Fanuc TP program (LS listing): FM112728.ls

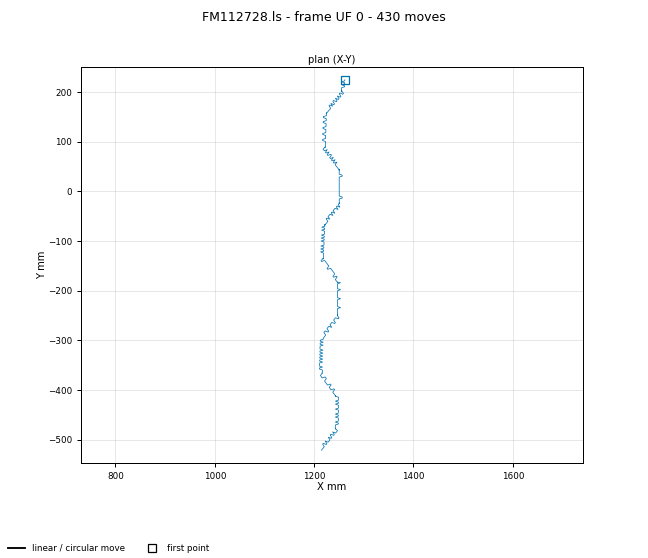
[picture p0: tool path of FM112728.ls in frame UF 0, 430 of 430 moves have a stored position in this frame; points joined in program order, loops and branches not executed]
/PROG  FM112728
/ATTR
OWNER		= MNEDITOR;
COMMENT		= "Auto FANUC move";
PROG_SIZE	= 0;
CREATE		= DATE 26-05-06  TIME 11:27:28;
MODIFIED	= DATE 26-05-06  TIME 11:27:28;
FILE_NAME	= ;
VERSION		= 0;
LINE_COUNT	= 435;
MEMORY_SIZE	= 0;
PROTECT		= READ_WRITE;
TCD:  STACK_SIZE	= 0,
      TASK_PRIORITY	= 50,
      TIME_SLICE	= 0,
      BUSY_LAMP_OFF	= 0,
      ABORT_REQUEST	= 0,
      PAUSE_REQUEST	= 0;
DEFAULT_GROUP	= 1,*,*,*,*;
CONTROL_CODE	= 00000000 00000000;
/MN
   1:  UFRAME_NUM=0 ;
   2:  UTOOL_NUM=1 ;
   3:  R[93]=10 ;
   4:  L P[1] 7mm/sec FINE ;
   5:  L P[2] 7mm/sec CNT50 ;
   6:  L P[3] 7mm/sec CNT50 ;
   7:  L P[4] 7mm/sec CNT50 ;
   8:  L P[5] 7mm/sec CNT50 ;
   9:  L P[6] 7mm/sec CNT50 ;
  10:  L P[7] 7mm/sec CNT50 ;
  11:  L P[8] 7mm/sec CNT50 ;
  12:  L P[9] 7mm/sec CNT50 ;
  13:  L P[10] 7mm/sec CNT50 ;
  14:  L P[11] 7mm/sec CNT50 ;
  15:  L P[12] 7mm/sec CNT50 ;
  16:  L P[13] 7mm/sec CNT50 ;
  17:  L P[14] 7mm/sec CNT50 ;
  18:  L P[15] 7mm/sec CNT50 ;
  19:  L P[16] 7mm/sec CNT50 ;
  20:  L P[17] 7mm/sec CNT50 ;
  21:  L P[18] 7mm/sec CNT50 ;
  22:  L P[19] 7mm/sec CNT50 ;
  23:  L P[20] 7mm/sec CNT50 ;
  24:  L P[21] 7mm/sec CNT50 ;
  25:  L P[22] 7mm/sec CNT50 ;
  26:  L P[23] 7mm/sec CNT50 ;
  27:  L P[24] 7mm/sec CNT50 ;
  28:  L P[25] 7mm/sec CNT50 ;
  29:  L P[26] 7mm/sec CNT50 ;
  30:  L P[27] 7mm/sec CNT50 ;
  31:  L P[28] 7mm/sec CNT50 ;
  32:  L P[29] 7mm/sec CNT50 ;
  33:  L P[30] 7mm/sec CNT50 ;
  34:  L P[31] 7mm/sec CNT50 ;
  35:  L P[32] 7mm/sec CNT50 ;
  36:  L P[33] 7mm/sec CNT50 ;
  37:  L P[34] 7mm/sec CNT50 ;
  38:  L P[35] 7mm/sec CNT50 ;
  39:  L P[36] 7mm/sec CNT50 ;
  40:  L P[37] 7mm/sec CNT50 ;
  41:  L P[38] 7mm/sec CNT50 ;
  42:  L P[39] 7mm/sec CNT50 ;
  43:  L P[40] 7mm/sec CNT50 ;
  44:  L P[41] 7mm/sec CNT50 ;
  45:  L P[42] 7mm/sec CNT50 ;
  46:  L P[43] 7mm/sec CNT50 ;
  47:  L P[44] 7mm/sec CNT50 ;
  48:  L P[45] 7mm/sec CNT50 ;
  49:  L P[46] 7mm/sec CNT50 ;
  50:  L P[47] 7mm/sec CNT50 ;
  51:  L P[48] 7mm/sec CNT50 ;
  52:  L P[49] 7mm/sec CNT50 ;
  53:  L P[50] 7mm/sec CNT50 ;
  54:  L P[51] 7mm/sec CNT50 ;
  55:  L P[52] 7mm/sec CNT50 ;
  56:  L P[53] 7mm/sec CNT50 ;
  57:  L P[54] 7mm/sec CNT50 ;
  58:  L P[55] 7mm/sec CNT50 ;
  59:  L P[56] 7mm/sec CNT50 ;
  60:  L P[57] 7mm/sec CNT50 ;
  61:  L P[58] 7mm/sec CNT50 ;
  62:  L P[59] 7mm/sec CNT50 ;
  63:  L P[60] 7mm/sec CNT50 ;
  64:  L P[61] 7mm/sec CNT50 ;
  65:  L P[62] 7mm/sec CNT50 ;
  66:  L P[63] 7mm/sec CNT50 ;
  67:  L P[64] 7mm/sec CNT50 ;
  68:  L P[65] 7mm/sec CNT50 ;
  69:  L P[66] 7mm/sec CNT50 ;
  70:  L P[67] 7mm/sec CNT50 ;
  71:  L P[68] 7mm/sec CNT50 ;
  72:  L P[69] 7mm/sec CNT50 ;
  73:  L P[70] 7mm/sec CNT50 ;
  74:  L P[71] 7mm/sec CNT50 ;
  75:  L P[72] 7mm/sec CNT50 ;
  76:  L P[73] 7mm/sec CNT50 ;
  77:  L P[74] 7mm/sec CNT50 ;
  78:  L P[75] 7mm/sec CNT50 ;
  79:  L P[76] 7mm/sec CNT50 ;
  80:  L P[77] 7mm/sec CNT50 ;
  81:  L P[78] 7mm/sec CNT50 ;
  82:  L P[79] 7mm/sec CNT50 ;
  83:  L P[80] 7mm/sec CNT50 ;
  84:  L P[81] 7mm/sec CNT50 ;
  85:  L P[82] 7mm/sec CNT50 ;
  86:  L P[83] 7mm/sec CNT50 ;
  87:  L P[84] 7mm/sec CNT50 ;
  88:  L P[85] 7mm/sec CNT50 ;
  89:  L P[86] 7mm/sec CNT50 ;
  90:  L P[87] 7mm/sec CNT50 ;
  91:  L P[88] 7mm/sec CNT50 ;
  92:  L P[89] 7mm/sec CNT50 ;
  93:  L P[90] 7mm/sec CNT50 ;
  94:  L P[91] 7mm/sec CNT50 ;
  95:  L P[92] 7mm/sec CNT50 ;
  96:  L P[93] 7mm/sec CNT50 ;
  97:  L P[94] 7mm/sec CNT50 ;
  98:  L P[95] 7mm/sec CNT50 ;
  99:  L P[96] 7mm/sec CNT50 ;
 100:  L P[97] 7mm/sec CNT50 ;
 101:  L P[98] 7mm/sec CNT50 ;
 102:  L P[99] 7mm/sec CNT50 ;
 103:  L P[100] 7mm/sec CNT50 ;
 104:  L P[101] 7mm/sec CNT50 ;
 105:  L P[102] 7mm/sec CNT50 ;
 106:  L P[103] 7mm/sec CNT50 ;
 107:  L P[104] 7mm/sec CNT50 ;
 108:  L P[105] 7mm/sec CNT50 ;
 109:  L P[106] 7mm/sec CNT50 ;
 110:  L P[107] 7mm/sec CNT50 ;
 111:  L P[108] 7mm/sec CNT50 ;
 112:  L P[109] 7mm/sec CNT50 ;
 113:  L P[110] 7mm/sec CNT50 ;
 114:  L P[111] 7mm/sec CNT50 ;
 115:  L P[112] 7mm/sec CNT50 ;
 116:  L P[113] 7mm/sec CNT50 ;
 117:  L P[114] 7mm/sec CNT50 ;
 118:  L P[115] 7mm/sec CNT50 ;
 119:  L P[116] 7mm/sec CNT50 ;
 120:  L P[117] 7mm/sec CNT50 ;
 121:  L P[118] 7mm/sec CNT50 ;
 122:  L P[119] 7mm/sec CNT50 ;
 123:  L P[120] 7mm/sec CNT50 ;
 124:  L P[121] 7mm/sec CNT50 ;
 125:  L P[122] 7mm/sec CNT50 ;
 126:  L P[123] 7mm/sec CNT50 ;
 127:  L P[124] 7mm/sec CNT50 ;
 128:  L P[125] 7mm/sec CNT50 ;
 129:  L P[126] 7mm/sec CNT50 ;
 130:  L P[127] 7mm/sec CNT50 ;
 131:  L P[128] 7mm/sec CNT50 ;
 132:  L P[129] 7mm/sec CNT50 ;
 133:  L P[130] 7mm/sec CNT50 ;
 134:  L P[131] 7mm/sec CNT50 ;
 135:  L P[132] 7mm/sec CNT50 ;
 136:  L P[133] 7mm/sec CNT50 ;
 137:  L P[134] 7mm/sec CNT50 ;
 138:  L P[135] 7mm/sec CNT50 ;
 139:  L P[136] 7mm/sec CNT50 ;
 140:  L P[137] 7mm/sec CNT50 ;
 141:  L P[138] 7mm/sec CNT50 ;
 142:  L P[139] 7mm/sec CNT50 ;
 143:  L P[140] 7mm/sec CNT50 ;
 144:  L P[141] 7mm/sec CNT50 ;
 145:  L P[142] 7mm/sec CNT50 ;
 146:  L P[143] 7mm/sec CNT50 ;
 147:  L P[144] 7mm/sec CNT50 ;
 148:  L P[145] 7mm/sec CNT50 ;
 149:  L P[146] 7mm/sec CNT50 ;
 150:  L P[147] 7mm/sec CNT50 ;
 151:  L P[148] 7mm/sec CNT50 ;
 152:  L P[149] 7mm/sec CNT50 ;
 153:  L P[150] 7mm/sec CNT50 ;
 154:  L P[151] 7mm/sec CNT50 ;
 155:  L P[152] 7mm/sec CNT50 ;
 156:  L P[153] 7mm/sec CNT50 ;
 157:  L P[154] 7mm/sec CNT50 ;
 158:  L P[155] 7mm/sec CNT50 ;
 159:  L P[156] 7mm/sec CNT50 ;
 160:  L P[157] 7mm/sec CNT50 ;
 161:  L P[158] 7mm/sec CNT50 ;
 162:  L P[159] 7mm/sec CNT50 ;
 163:  L P[160] 7mm/sec CNT50 ;
 164:  L P[161] 7mm/sec CNT50 ;
 165:  L P[162] 7mm/sec CNT50 ;
 166:  L P[163] 7mm/sec CNT50 ;
 167:  L P[164] 7mm/sec CNT50 ;
 168:  L P[165] 7mm/sec CNT50 ;
 169:  L P[166] 7mm/sec CNT50 ;
 170:  L P[167] 7mm/sec CNT50 ;
 171:  L P[168] 7mm/sec CNT50 ;
 172:  L P[169] 7mm/sec CNT50 ;
 173:  L P[170] 7mm/sec CNT50 ;
 174:  L P[171] 7mm/sec CNT50 ;
 175:  L P[172] 7mm/sec CNT50 ;
 176:  L P[173] 7mm/sec CNT50 ;
 177:  L P[174] 7mm/sec CNT50 ;
 178:  L P[175] 7mm/sec CNT50 ;
 179:  L P[176] 7mm/sec CNT50 ;
 180:  L P[177] 7mm/sec CNT50 ;
 181:  L P[178] 7mm/sec CNT50 ;
 182:  L P[179] 7mm/sec CNT50 ;
 183:  L P[180] 7mm/sec CNT50 ;
 184:  L P[181] 7mm/sec CNT50 ;
 185:  L P[182] 7mm/sec CNT50 ;
 186:  L P[183] 7mm/sec CNT50 ;
 187:  L P[184] 7mm/sec CNT50 ;
 188:  L P[185] 7mm/sec CNT50 ;
 189:  L P[186] 7mm/sec CNT50 ;
 190:  L P[187] 7mm/sec CNT50 ;
 191:  L P[188] 7mm/sec CNT50 ;
 192:  L P[189] 7mm/sec CNT50 ;
 193:  L P[190] 7mm/sec CNT50 ;
 194:  L P[191] 7mm/sec CNT50 ;
 195:  L P[192] 7mm/sec CNT50 ;
 196:  L P[193] 7mm/sec CNT50 ;
 197:  L P[194] 7mm/sec CNT50 ;
 198:  L P[195] 7mm/sec CNT50 ;
 199:  L P[196] 7mm/sec CNT50 ;
 200:  L P[197] 7mm/sec CNT50 ;
 201:  L P[198] 7mm/sec CNT50 ;
 202:  L P[199] 7mm/sec CNT50 ;
 203:  L P[200] 7mm/sec CNT50 ;
 204:  L P[201] 7mm/sec CNT50 ;
 205:  L P[202] 7mm/sec CNT50 ;
 206:  L P[203] 7mm/sec CNT50 ;
 207:  L P[204] 7mm/sec CNT50 ;
 208:  L P[205] 7mm/sec CNT50 ;
 209:  L P[206] 7mm/sec CNT50 ;
 210:  L P[207] 7mm/sec CNT50 ;
 211:  L P[208] 7mm/sec CNT50 ;
 212:  L P[209] 7mm/sec CNT50 ;
 213:  L P[210] 7mm/sec CNT50 ;
 214:  L P[211] 7mm/sec CNT50 ;
 215:  L P[212] 7mm/sec CNT50 ;
 216:  L P[213] 7mm/sec CNT50 ;
 217:  L P[214] 7mm/sec CNT50 ;
 218:  L P[215] 7mm/sec CNT50 ;
 219:  L P[216] 7mm/sec CNT50 ;
 220:  L P[217] 7mm/sec CNT50 ;
 221:  L P[218] 7mm/sec CNT50 ;
 222:  L P[219] 7mm/sec CNT50 ;
 223:  L P[220] 7mm/sec CNT50 ;
 224:  L P[221] 7mm/sec CNT50 ;
 225:  L P[222] 7mm/sec CNT50 ;
 226:  L P[223] 7mm/sec CNT50 ;
 227:  L P[224] 7mm/sec CNT50 ;
 228:  L P[225] 7mm/sec CNT50 ;
 229:  L P[226] 7mm/sec CNT50 ;
 230:  L P[227] 7mm/sec CNT50 ;
 231:  L P[228] 7mm/sec CNT50 ;
 232:  L P[229] 7mm/sec CNT50 ;
 233:  L P[230] 7mm/sec CNT50 ;
 234:  L P[231] 7mm/sec CNT50 ;
 235:  L P[232] 7mm/sec CNT50 ;
 236:  L P[233] 7mm/sec CNT50 ;
 237:  L P[234] 7mm/sec CNT50 ;
 238:  L P[235] 7mm/sec CNT50 ;
 239:  L P[236] 7mm/sec CNT50 ;
 240:  L P[237] 7mm/sec CNT50 ;
 241:  L P[238] 7mm/sec CNT50 ;
 242:  L P[239] 7mm/sec CNT50 ;
 243:  L P[240] 7mm/sec CNT50 ;
 244:  L P[241] 7mm/sec CNT50 ;
 245:  L P[242] 7mm/sec CNT50 ;
 246:  L P[243] 7mm/sec CNT50 ;
 247:  L P[244] 7mm/sec CNT50 ;
 248:  L P[245] 7mm/sec CNT50 ;
 249:  L P[246] 7mm/sec CNT50 ;
 250:  L P[247] 7mm/sec CNT50 ;
 251:  L P[248] 7mm/sec CNT50 ;
 252:  L P[249] 7mm/sec CNT50 ;
 253:  L P[250] 7mm/sec CNT50 ;
 254:  L P[251] 7mm/sec CNT50 ;
 255:  L P[252] 7mm/sec CNT50 ;
 256:  L P[253] 7mm/sec CNT50 ;
 257:  L P[254] 7mm/sec CNT50 ;
 258:  L P[255] 7mm/sec CNT50 ;
 259:  L P[256] 7mm/sec CNT50 ;
 260:  L P[257] 7mm/sec CNT50 ;
 261:  L P[258] 7mm/sec CNT50 ;
 262:  L P[259] 7mm/sec CNT50 ;
 263:  L P[260] 7mm/sec CNT50 ;
 264:  L P[261] 7mm/sec CNT50 ;
 265:  L P[262] 7mm/sec CNT50 ;
 266:  L P[263] 7mm/sec CNT50 ;
 267:  L P[264] 7mm/sec CNT50 ;
 268:  L P[265] 7mm/sec CNT50 ;
 269:  L P[266] 7mm/sec CNT50 ;
 270:  L P[267] 7mm/sec CNT50 ;
 271:  L P[268] 7mm/sec CNT50 ;
 272:  L P[269] 7mm/sec CNT50 ;
 273:  L P[270] 7mm/sec CNT50 ;
 274:  L P[271] 7mm/sec CNT50 ;
 275:  L P[272] 7mm/sec CNT50 ;
 276:  L P[273] 7mm/sec CNT50 ;
 277:  L P[274] 7mm/sec CNT50 ;
 278:  L P[275] 7mm/sec CNT50 ;
 279:  L P[276] 7mm/sec CNT50 ;
 280:  L P[277] 7mm/sec CNT50 ;
 281:  L P[278] 7mm/sec CNT50 ;
 282:  L P[279] 7mm/sec CNT50 ;
 283:  L P[280] 7mm/sec CNT50 ;
 284:  L P[281] 7mm/sec CNT50 ;
 285:  L P[282] 7mm/sec CNT50 ;
 286:  L P[283] 7mm/sec CNT50 ;
 287:  L P[284] 7mm/sec CNT50 ;
 288:  L P[285] 7mm/sec CNT50 ;
 289:  L P[286] 7mm/sec CNT50 ;
 290:  L P[287] 7mm/sec CNT50 ;
 291:  L P[288] 7mm/sec CNT50 ;
 292:  L P[289] 7mm/sec CNT50 ;
 293:  L P[290] 7mm/sec CNT50 ;
 294:  L P[291] 7mm/sec CNT50 ;
 295:  L P[292] 7mm/sec CNT50 ;
 296:  L P[293] 7mm/sec CNT50 ;
 297:  L P[294] 7mm/sec CNT50 ;
 298:  L P[295] 7mm/sec CNT50 ;
 299:  L P[296] 7mm/sec CNT50 ;
 300:  L P[297] 7mm/sec CNT50 ;
 301:  L P[298] 7mm/sec CNT50 ;
 302:  L P[299] 7mm/sec CNT50 ;
 303:  L P[300] 7mm/sec CNT50 ;
 304:  L P[301] 7mm/sec CNT50 ;
 305:  L P[302] 7mm/sec CNT50 ;
 306:  L P[303] 7mm/sec CNT50 ;
 307:  L P[304] 7mm/sec CNT50 ;
 308:  L P[305] 7mm/sec CNT50 ;
 309:  L P[306] 7mm/sec CNT50 ;
 310:  L P[307] 7mm/sec CNT50 ;
 311:  L P[308] 7mm/sec CNT50 ;
 312:  L P[309] 7mm/sec CNT50 ;
 313:  L P[310] 7mm/sec CNT50 ;
 314:  L P[311] 7mm/sec CNT50 ;
 315:  L P[312] 7mm/sec CNT50 ;
 316:  L P[313] 7mm/sec CNT50 ;
 317:  L P[314] 7mm/sec CNT50 ;
 318:  L P[315] 7mm/sec CNT50 ;
 319:  L P[316] 7mm/sec CNT50 ;
 320:  L P[317] 7mm/sec CNT50 ;
 321:  L P[318] 7mm/sec CNT50 ;
 322:  L P[319] 7mm/sec CNT50 ;
 323:  L P[320] 7mm/sec CNT50 ;
 324:  L P[321] 7mm/sec CNT50 ;
 325:  L P[322] 7mm/sec CNT50 ;
 326:  L P[323] 7mm/sec CNT50 ;
 327:  L P[324] 7mm/sec CNT50 ;
 328:  L P[325] 7mm/sec CNT50 ;
 329:  L P[326] 7mm/sec CNT50 ;
 330:  L P[327] 7mm/sec CNT50 ;
 331:  L P[328] 7mm/sec CNT50 ;
 332:  L P[329] 7mm/sec CNT50 ;
 333:  L P[330] 7mm/sec CNT50 ;
 334:  L P[331] 7mm/sec CNT50 ;
 335:  L P[332] 7mm/sec CNT50 ;
 336:  L P[333] 7mm/sec CNT50 ;
 337:  L P[334] 7mm/sec CNT50 ;
 338:  L P[335] 7mm/sec CNT50 ;
 339:  L P[336] 7mm/sec CNT50 ;
 340:  L P[337] 7mm/sec CNT50 ;
 341:  L P[338] 7mm/sec CNT50 ;
 342:  L P[339] 7mm/sec CNT50 ;
 343:  L P[340] 7mm/sec CNT50 ;
 344:  L P[341] 7mm/sec CNT50 ;
 345:  L P[342] 7mm/sec CNT50 ;
 346:  L P[343] 7mm/sec CNT50 ;
 347:  L P[344] 7mm/sec CNT50 ;
 348:  L P[345] 7mm/sec CNT50 ;
 349:  L P[346] 7mm/sec CNT50 ;
 350:  L P[347] 7mm/sec CNT50 ;
 351:  L P[348] 7mm/sec CNT50 ;
 352:  L P[349] 7mm/sec CNT50 ;
 353:  L P[350] 7mm/sec CNT50 ;
 354:  L P[351] 7mm/sec CNT50 ;
 355:  L P[352] 7mm/sec CNT50 ;
 356:  L P[353] 7mm/sec CNT50 ;
 357:  L P[354] 7mm/sec CNT50 ;
 358:  L P[355] 7mm/sec CNT50 ;
 359:  L P[356] 7mm/sec CNT50 ;
 360:  L P[357] 7mm/sec CNT50 ;
 361:  L P[358] 7mm/sec CNT50 ;
 362:  L P[359] 7mm/sec CNT50 ;
 363:  L P[360] 7mm/sec CNT50 ;
 364:  L P[361] 7mm/sec CNT50 ;
 365:  L P[362] 7mm/sec CNT50 ;
 366:  L P[363] 7mm/sec CNT50 ;
 367:  L P[364] 7mm/sec CNT50 ;
 368:  L P[365] 7mm/sec CNT50 ;
 369:  L P[366] 7mm/sec CNT50 ;
 370:  L P[367] 7mm/sec CNT50 ;
 371:  L P[368] 7mm/sec CNT50 ;
 372:  L P[369] 7mm/sec CNT50 ;
 373:  L P[370] 7mm/sec CNT50 ;
 374:  L P[371] 7mm/sec CNT50 ;
 375:  L P[372] 7mm/sec CNT50 ;
 376:  L P[373] 7mm/sec CNT50 ;
 377:  L P[374] 7mm/sec CNT50 ;
 378:  L P[375] 7mm/sec CNT50 ;
 379:  L P[376] 7mm/sec CNT50 ;
 380:  L P[377] 7mm/sec CNT50 ;
 381:  L P[378] 7mm/sec CNT50 ;
 382:  L P[379] 7mm/sec CNT50 ;
 383:  L P[380] 7mm/sec CNT50 ;
 384:  L P[381] 7mm/sec CNT50 ;
 385:  L P[382] 7mm/sec CNT50 ;
 386:  L P[383] 7mm/sec CNT50 ;
 387:  L P[384] 7mm/sec CNT50 ;
 388:  L P[385] 7mm/sec CNT50 ;
 389:  L P[386] 7mm/sec CNT50 ;
 390:  L P[387] 7mm/sec CNT50 ;
 391:  L P[388] 7mm/sec CNT50 ;
 392:  L P[389] 7mm/sec CNT50 ;
 393:  L P[390] 7mm/sec CNT50 ;
 394:  L P[391] 7mm/sec CNT50 ;
 395:  L P[392] 7mm/sec CNT50 ;
 396:  L P[393] 7mm/sec CNT50 ;
 397:  L P[394] 7mm/sec CNT50 ;
 398:  L P[395] 7mm/sec CNT50 ;
 399:  L P[396] 7mm/sec CNT50 ;
 400:  L P[397] 7mm/sec CNT50 ;
 401:  L P[398] 7mm/sec CNT50 ;
 402:  L P[399] 7mm/sec CNT50 ;
 403:  L P[400] 7mm/sec CNT50 ;
 404:  L P[401] 7mm/sec CNT50 ;
 405:  L P[402] 7mm/sec CNT50 ;
 406:  L P[403] 7mm/sec CNT50 ;
 407:  L P[404] 7mm/sec CNT50 ;
 408:  L P[405] 7mm/sec CNT50 ;
 409:  L P[406] 7mm/sec CNT50 ;
 410:  L P[407] 7mm/sec CNT50 ;
 411:  L P[408] 7mm/sec CNT50 ;
 412:  L P[409] 7mm/sec CNT50 ;
 413:  L P[410] 7mm/sec CNT50 ;
 414:  L P[411] 7mm/sec CNT50 ;
 415:  L P[412] 7mm/sec CNT50 ;
 416:  L P[413] 7mm/sec CNT50 ;
 417:  L P[414] 7mm/sec CNT50 ;
 418:  L P[415] 7mm/sec CNT50 ;
 419:  L P[416] 7mm/sec CNT50 ;
 420:  L P[417] 7mm/sec CNT50 ;
 421:  L P[418] 7mm/sec CNT50 ;
 422:  L P[419] 7mm/sec CNT50 ;
 423:  L P[420] 7mm/sec CNT50 ;
 424:  L P[421] 7mm/sec CNT50 ;
 425:  L P[422] 7mm/sec CNT50 ;
 426:  L P[423] 7mm/sec CNT50 ;
 427:  L P[424] 7mm/sec CNT50 ;
 428:  L P[425] 7mm/sec CNT50 ;
 429:  L P[426] 7mm/sec CNT50 ;
 430:  L P[427] 7mm/sec CNT50 ;
 431:  L P[428] 7mm/sec CNT50 ;
 432:  L P[429] 7mm/sec CNT50 ;
 433:  L P[430] 7mm/sec FINE ;
 434:  R[93]=1 ;
 435:  END ;
/POS
P[1]{
   GP1:
	UF : 0, UT : 1,		CONFIG : 'N U T, 0, 0, 0',
	X = 1261.683  mm,	Y = 224.761  mm,	Z = -244.721  mm,
	W = 0.000 deg,	P = 30.000 deg,	R = 178.350 deg
};
P[2]{
   GP1:
	UF : 0, UT : 1,		CONFIG : 'N U T, 0, 0, 0',
	X = 1261.625  mm,	Y = 222.762  mm,	Z = -244.735  mm,
	W = 0.000 deg,	P = 30.000 deg,	R = 178.350 deg
};
P[3]{
   GP1:
	UF : 0, UT : 1,		CONFIG : 'N U T, 0, 0, 0',
	X = 1255.570  mm,	Y = 220.935  mm,	Z = -244.749  mm,
	W = 0.000 deg,	P = 30.000 deg,	R = 178.350 deg
};
P[4]{
   GP1:
	UF : 0, UT : 1,		CONFIG : 'N U T, 0, 0, 0',
	X = 1261.510  mm,	Y = 218.763  mm,	Z = -244.763  mm,
	W = 0.000 deg,	P = 30.000 deg,	R = 178.350 deg
};
P[5]{
   GP1:
	UF : 0, UT : 1,		CONFIG : 'N U T, 0, 0, 0',
	X = 1261.452  mm,	Y = 216.764  mm,	Z = -244.777  mm,
	W = 0.000 deg,	P = 30.000 deg,	R = 178.350 deg
};
P[6]{
   GP1:
	UF : 0, UT : 1,		CONFIG : 'N U T, 0, 0, 0',
	X = 1255.397  mm,	Y = 214.938  mm,	Z = -244.792  mm,
	W = 0.000 deg,	P = 30.000 deg,	R = 178.350 deg
};
P[7]{
   GP1:
	UF : 0, UT : 1,		CONFIG : 'N U T, 0, 0, 0',
	X = 1261.337  mm,	Y = 212.766  mm,	Z = -244.806  mm,
	W = 0.000 deg,	P = 30.000 deg,	R = 178.350 deg
};
P[8]{
   GP1:
	UF : 0, UT : 1,		CONFIG : 'N U T, 0, 0, 0',
	X = 1261.280  mm,	Y = 210.767  mm,	Z = -244.820  mm,
	W = 0.000 deg,	P = 30.000 deg,	R = 178.350 deg
};
P[9]{
   GP1:
	UF : 0, UT : 1,		CONFIG : 'N U T, 0, 0, 0',
	X = 1255.224  mm,	Y = 208.940  mm,	Z = -244.834  mm,
	W = 0.000 deg,	P = 30.000 deg,	R = 170.556 deg
};
P[10]{
   GP1:
	UF : 0, UT : 1,		CONFIG : 'N U T, 0, 0, 0',
	X = 1255.167  mm,	Y = 206.941  mm,	Z = -244.848  mm,
	W = 0.000 deg,	P = 30.000 deg,	R = 162.762 deg
};
P[11]{
   GP1:
	UF : 0, UT : 1,		CONFIG : 'N U T, 0, 0, 0',
	X = 1255.109  mm,	Y = 204.942  mm,	Z = -244.862  mm,
	W = 0.000 deg,	P = 30.000 deg,	R = 154.967 deg
};
P[12]{
   GP1:
	UF : 0, UT : 1,		CONFIG : 'N U T, 0, 0, 0',
	X = 1255.052  mm,	Y = 202.943  mm,	Z = -244.877  mm,
	W = 0.000 deg,	P = 30.000 deg,	R = 147.173 deg
};
P[13]{
   GP1:
	UF : 0, UT : 1,		CONFIG : 'N U T, 0, 0, 0',
	X = 1254.994  mm,	Y = 200.944  mm,	Z = -244.891  mm,
	W = 0.000 deg,	P = 30.000 deg,	R = 139.379 deg
};
P[14]{
   GP1:
	UF : 0, UT : 1,		CONFIG : 'N U T, 0, 0, 0',
	X = 1255.605  mm,	Y = 202.508  mm,	Z = -244.892  mm,
	W = 0.000 deg,	P = 30.000 deg,	R = 139.379 deg
};
P[15]{
   GP1:
	UF : 0, UT : 1,		CONFIG : 'N U T, 0, 0, 0',
	X = 1259.086  mm,	Y = 197.357  mm,	Z = -244.654  mm,
	W = 0.000 deg,	P = 30.000 deg,	R = 139.379 deg
};
P[16]{
   GP1:
	UF : 0, UT : 1,		CONFIG : 'N U T, 0, 0, 0',
	X = 1257.795  mm,	Y = 195.851  mm,	Z = -244.393  mm,
	W = 0.000 deg,	P = 30.000 deg,	R = 139.379 deg
};
P[17]{
   GP1:
	UF : 0, UT : 1,		CONFIG : 'N U T, 0, 0, 0',
	X = 1251.949  mm,	Y = 198.253  mm,	Z = -244.133  mm,
	W = 0.000 deg,	P = 30.000 deg,	R = 139.379 deg
};
P[18]{
   GP1:
	UF : 0, UT : 1,		CONFIG : 'N U T, 0, 0, 0',
	X = 1250.658  mm,	Y = 196.748  mm,	Z = -243.872  mm,
	W = 0.000 deg,	P = 30.000 deg,	R = 139.379 deg
};
P[19]{
   GP1:
	UF : 0, UT : 1,		CONFIG : 'N U T, 0, 0, 0',
	X = 1253.922  mm,	Y = 191.336  mm,	Z = -243.612  mm,
	W = 0.000 deg,	P = 30.000 deg,	R = 139.379 deg
};
P[20]{
   GP1:
	UF : 0, UT : 1,		CONFIG : 'N U T, 0, 0, 0',
	X = 1252.631  mm,	Y = 189.831  mm,	Z = -243.351  mm,
	W = 0.000 deg,	P = 30.000 deg,	R = 139.379 deg
};
P[21]{
   GP1:
	UF : 0, UT : 1,		CONFIG : 'N U T, 0, 0, 0',
	X = 1246.785  mm,	Y = 192.232  mm,	Z = -243.090  mm,
	W = 0.000 deg,	P = 30.000 deg,	R = 139.379 deg
};
P[22]{
   GP1:
	UF : 0, UT : 1,		CONFIG : 'N U T, 0, 0, 0',
	X = 1250.049  mm,	Y = 186.821  mm,	Z = -242.830  mm,
	W = 0.000 deg,	P = 30.000 deg,	R = 139.379 deg
};
P[23]{
   GP1:
	UF : 0, UT : 1,		CONFIG : 'N U T, 0, 0, 0',
	X = 1248.758  mm,	Y = 185.316  mm,	Z = -242.569  mm,
	W = 0.000 deg,	P = 30.000 deg,	R = 139.379 deg
};
P[24]{
   GP1:
	UF : 0, UT : 1,		CONFIG : 'N U T, 0, 0, 0',
	X = 1242.912  mm,	Y = 187.717  mm,	Z = -242.309  mm,
	W = 0.000 deg,	P = 30.000 deg,	R = 139.379 deg
};
P[25]{
   GP1:
	UF : 0, UT : 1,		CONFIG : 'N U T, 0, 0, 0',
	X = 1246.176  mm,	Y = 182.305  mm,	Z = -242.048  mm,
	W = 0.000 deg,	P = 30.000 deg,	R = 139.379 deg
};
P[26]{
   GP1:
	UF : 0, UT : 1,		CONFIG : 'N U T, 0, 0, 0',
	X = 1244.885  mm,	Y = 180.800  mm,	Z = -241.787  mm,
	W = 0.000 deg,	P = 30.000 deg,	R = 139.379 deg
};
P[27]{
   GP1:
	UF : 0, UT : 1,		CONFIG : 'N U T, 0, 0, 0',
	X = 1239.039  mm,	Y = 183.201  mm,	Z = -241.527  mm,
	W = 0.000 deg,	P = 30.000 deg,	R = 139.379 deg
};
P[28]{
   GP1:
	UF : 0, UT : 1,		CONFIG : 'N U T, 0, 0, 0',
	X = 1237.748  mm,	Y = 181.696  mm,	Z = -241.266  mm,
	W = 0.000 deg,	P = 30.000 deg,	R = 139.379 deg
};
P[29]{
   GP1:
	UF : 0, UT : 1,		CONFIG : 'N U T, 0, 0, 0',
	X = 1241.012  mm,	Y = 176.285  mm,	Z = -241.006  mm,
	W = 0.000 deg,	P = 30.000 deg,	R = 139.379 deg
};
P[30]{
   GP1:
	UF : 0, UT : 1,		CONFIG : 'N U T, 0, 0, 0',
	X = 1239.721  mm,	Y = 174.780  mm,	Z = -240.745  mm,
	W = 0.000 deg,	P = 30.000 deg,	R = 139.379 deg
};
P[31]{
   GP1:
	UF : 0, UT : 1,		CONFIG : 'N U T, 0, 0, 0',
	X = 1233.875  mm,	Y = 177.181  mm,	Z = -240.484  mm,
	W = 0.000 deg,	P = 30.000 deg,	R = 139.379 deg
};
P[32]{
   GP1:
	UF : 0, UT : 1,		CONFIG : 'N U T, 0, 0, 0',
	X = 1237.139  mm,	Y = 171.770  mm,	Z = -240.224  mm,
	W = 0.000 deg,	P = 30.000 deg,	R = 139.379 deg
};
P[33]{
   GP1:
	UF : 0, UT : 1,		CONFIG : 'N U T, 0, 0, 0',
	X = 1231.293  mm,	Y = 174.171  mm,	Z = -239.963  mm,
	W = 0.000 deg,	P = 30.000 deg,	R = 139.379 deg
};
P[34]{
   GP1:
	UF : 0, UT : 1,		CONFIG : 'N U T, 0, 0, 0',
	X = 1230.002  mm,	Y = 172.666  mm,	Z = -239.703  mm,
	W = 0.000 deg,	P = 30.000 deg,	R = 139.379 deg
};
P[35]{
   GP1:
	UF : 0, UT : 1,		CONFIG : 'N U T, 0, 0, 0',
	X = 1233.266  mm,	Y = 167.254  mm,	Z = -239.442  mm,
	W = 0.000 deg,	P = 30.000 deg,	R = 139.379 deg
};
P[36]{
   GP1:
	UF : 0, UT : 1,		CONFIG : 'N U T, 0, 0, 0',
	X = 1231.974  mm,	Y = 165.749  mm,	Z = -239.181  mm,
	W = 0.000 deg,	P = 30.000 deg,	R = 139.379 deg
};
P[37]{
   GP1:
	UF : 0, UT : 1,		CONFIG : 'N U T, 0, 0, 0',
	X = 1230.683  mm,	Y = 164.244  mm,	Z = -238.921  mm,
	W = 0.000 deg,	P = 30.000 deg,	R = 146.431 deg
};
P[38]{
   GP1:
	UF : 0, UT : 1,		CONFIG : 'N U T, 0, 0, 0',
	X = 1229.392  mm,	Y = 162.739  mm,	Z = -238.660  mm,
	W = 0.000 deg,	P = 30.000 deg,	R = 154.151 deg
};
P[39]{
   GP1:
	UF : 0, UT : 1,		CONFIG : 'N U T, 0, 0, 0',
	X = 1228.101  mm,	Y = 161.234  mm,	Z = -238.400  mm,
	W = 0.000 deg,	P = 30.000 deg,	R = 161.872 deg
};
P[40]{
   GP1:
	UF : 0, UT : 1,		CONFIG : 'N U T, 0, 0, 0',
	X = 1226.810  mm,	Y = 159.729  mm,	Z = -238.139  mm,
	W = 0.000 deg,	P = 30.000 deg,	R = 169.592 deg
};
P[41]{
   GP1:
	UF : 0, UT : 1,		CONFIG : 'N U T, 0, 0, 0',
	X = 1225.519  mm,	Y = 158.223  mm,	Z = -237.879  mm,
	W = 0.000 deg,	P = 30.000 deg,	R = 177.312 deg
};
P[42]{
   GP1:
	UF : 0, UT : 1,		CONFIG : 'N U T, 0, 0, 0',
	X = 1224.228  mm,	Y = 156.718  mm,	Z = -237.618  mm,
	W = 0.000 deg,	P = 30.000 deg,	R = 177.979 deg
};
P[43]{
   GP1:
	UF : 0, UT : 1,		CONFIG : 'N U T, 0, 0, 0',
	X = 1224.894  mm,	Y = 158.431  mm,	Z = -237.608  mm,
	W = 0.000 deg,	P = 30.000 deg,	R = 177.979 deg
};
P[44]{
   GP1:
	UF : 0, UT : 1,		CONFIG : 'N U T, 0, 0, 0',
	X = 1224.830  mm,	Y = 156.587  mm,	Z = -237.622  mm,
	W = 0.000 deg,	P = 30.000 deg,	R = 177.979 deg
};
P[45]{
   GP1:
	UF : 0, UT : 1,		CONFIG : 'N U T, 0, 0, 0',
	X = 1224.760  mm,	Y = 154.588  mm,	Z = -237.637  mm,
	W = 0.000 deg,	P = 30.000 deg,	R = 177.979 deg
};
P[46]{
   GP1:
	UF : 0, UT : 1,		CONFIG : 'N U T, 0, 0, 0',
	X = 1224.689  mm,	Y = 152.589  mm,	Z = -237.652  mm,
	W = 0.000 deg,	P = 30.000 deg,	R = 177.979 deg
};
P[47]{
   GP1:
	UF : 0, UT : 1,		CONFIG : 'N U T, 0, 0, 0',
	X = 1218.622  mm,	Y = 150.802  mm,	Z = -237.666  mm,
	W = 0.000 deg,	P = 30.000 deg,	R = 177.979 deg
};
P[48]{
   GP1:
	UF : 0, UT : 1,		CONFIG : 'N U T, 0, 0, 0',
	X = 1218.552  mm,	Y = 148.803  mm,	Z = -237.681  mm,
	W = 0.000 deg,	P = 30.000 deg,	R = 177.979 deg
};
P[49]{
   GP1:
	UF : 0, UT : 1,		CONFIG : 'N U T, 0, 0, 0',
	X = 1224.478  mm,	Y = 146.593  mm,	Z = -237.696  mm,
	W = 0.000 deg,	P = 30.000 deg,	R = 177.979 deg
};
P[50]{
   GP1:
	UF : 0, UT : 1,		CONFIG : 'N U T, 0, 0, 0',
	X = 1224.407  mm,	Y = 144.594  mm,	Z = -237.711  mm,
	W = 0.000 deg,	P = 30.000 deg,	R = 177.979 deg
};
P[51]{
   GP1:
	UF : 0, UT : 1,		CONFIG : 'N U T, 0, 0, 0',
	X = 1224.337  mm,	Y = 142.596  mm,	Z = -237.726  mm,
	W = 0.000 deg,	P = 30.000 deg,	R = 177.979 deg
};
P[52]{
   GP1:
	UF : 0, UT : 1,		CONFIG : 'N U T, 0, 0, 0',
	X = 1218.270  mm,	Y = 140.809  mm,	Z = -237.741  mm,
	W = 0.000 deg,	P = 30.000 deg,	R = 177.979 deg
};
P[53]{
   GP1:
	UF : 0, UT : 1,		CONFIG : 'N U T, 0, 0, 0',
	X = 1218.199  mm,	Y = 138.810  mm,	Z = -237.756  mm,
	W = 0.000 deg,	P = 30.000 deg,	R = 177.979 deg
};
P[54]{
   GP1:
	UF : 0, UT : 1,		CONFIG : 'N U T, 0, 0, 0',
	X = 1224.125  mm,	Y = 136.600  mm,	Z = -237.771  mm,
	W = 0.000 deg,	P = 30.000 deg,	R = 177.979 deg
};
P[55]{
   GP1:
	UF : 0, UT : 1,		CONFIG : 'N U T, 0, 0, 0',
	X = 1224.054  mm,	Y = 134.601  mm,	Z = -237.785  mm,
	W = 0.000 deg,	P = 30.000 deg,	R = 177.979 deg
};
P[56]{
   GP1:
	UF : 0, UT : 1,		CONFIG : 'N U T, 0, 0, 0',
	X = 1223.984  mm,	Y = 132.602  mm,	Z = -237.800  mm,
	W = 0.000 deg,	P = 30.000 deg,	R = 177.979 deg
};
P[57]{
   GP1:
	UF : 0, UT : 1,		CONFIG : 'N U T, 0, 0, 0',
	X = 1223.913  mm,	Y = 130.604  mm,	Z = -237.815  mm,
	W = 0.000 deg,	P = 30.000 deg,	R = 177.979 deg
};
P[58]{
   GP1:
	UF : 0, UT : 1,		CONFIG : 'N U T, 0, 0, 0',
	X = 1217.847  mm,	Y = 128.816  mm,	Z = -237.830  mm,
	W = 0.000 deg,	P = 30.000 deg,	R = 177.979 deg
};
P[59]{
   GP1:
	UF : 0, UT : 1,		CONFIG : 'N U T, 0, 0, 0',
	X = 1217.776  mm,	Y = 126.818  mm,	Z = -237.845  mm,
	W = 0.000 deg,	P = 30.000 deg,	R = 177.979 deg
};
P[60]{
   GP1:
	UF : 0, UT : 1,		CONFIG : 'N U T, 0, 0, 0',
	X = 1223.702  mm,	Y = 124.607  mm,	Z = -237.860  mm,
	W = 0.000 deg,	P = 30.000 deg,	R = 177.979 deg
};
P[61]{
   GP1:
	UF : 0, UT : 1,		CONFIG : 'N U T, 0, 0, 0',
	X = 1223.631  mm,	Y = 122.609  mm,	Z = -237.875  mm,
	W = 0.000 deg,	P = 30.000 deg,	R = 177.979 deg
};
P[62]{
   GP1:
	UF : 0, UT : 1,		CONFIG : 'N U T, 0, 0, 0',
	X = 1223.561  mm,	Y = 120.610  mm,	Z = -237.890  mm,
	W = 0.000 deg,	P = 30.000 deg,	R = 177.979 deg
};
P[63]{
   GP1:
	UF : 0, UT : 1,		CONFIG : 'N U T, 0, 0, 0',
	X = 1223.490  mm,	Y = 118.611  mm,	Z = -237.904  mm,
	W = 0.000 deg,	P = 30.000 deg,	R = 177.979 deg
};
P[64]{
   GP1:
	UF : 0, UT : 1,		CONFIG : 'N U T, 0, 0, 0',
	X = 1217.423  mm,	Y = 116.824  mm,	Z = -237.919  mm,
	W = 0.000 deg,	P = 30.000 deg,	R = 177.979 deg
};
P[65]{
   GP1:
	UF : 0, UT : 1,		CONFIG : 'N U T, 0, 0, 0',
	X = 1217.353  mm,	Y = 114.826  mm,	Z = -237.934  mm,
	W = 0.000 deg,	P = 30.000 deg,	R = 177.979 deg
};
P[66]{
   GP1:
	UF : 0, UT : 1,		CONFIG : 'N U T, 0, 0, 0',
	X = 1223.279  mm,	Y = 112.615  mm,	Z = -237.949  mm,
	W = 0.000 deg,	P = 30.000 deg,	R = 177.979 deg
};
P[67]{
   GP1:
	UF : 0, UT : 1,		CONFIG : 'N U T, 0, 0, 0',
	X = 1223.208  mm,	Y = 110.617  mm,	Z = -237.964  mm,
	W = 0.000 deg,	P = 30.000 deg,	R = 177.979 deg
};
P[68]{
   GP1:
	UF : 0, UT : 1,		CONFIG : 'N U T, 0, 0, 0',
	X = 1223.138  mm,	Y = 108.618  mm,	Z = -237.979  mm,
	W = 0.000 deg,	P = 30.000 deg,	R = 177.979 deg
};
P[69]{
   GP1:
	UF : 0, UT : 1,		CONFIG : 'N U T, 0, 0, 0',
	X = 1223.067  mm,	Y = 106.619  mm,	Z = -237.994  mm,
	W = 0.000 deg,	P = 30.000 deg,	R = 177.979 deg
};
P[70]{
   GP1:
	UF : 0, UT : 1,		CONFIG : 'N U T, 0, 0, 0',
	X = 1217.000  mm,	Y = 104.832  mm,	Z = -238.008  mm,
	W = 0.000 deg,	P = 30.000 deg,	R = 177.979 deg
};
P[71]{
   GP1:
	UF : 0, UT : 1,		CONFIG : 'N U T, 0, 0, 0',
	X = 1216.930  mm,	Y = 102.833  mm,	Z = -238.023  mm,
	W = 0.000 deg,	P = 30.000 deg,	R = 177.979 deg
};
P[72]{
   GP1:
	UF : 0, UT : 1,		CONFIG : 'N U T, 0, 0, 0',
	X = 1222.855  mm,	Y = 100.623  mm,	Z = -238.038  mm,
	W = 0.000 deg,	P = 30.000 deg,	R = 177.979 deg
};
P[73]{
   GP1:
	UF : 0, UT : 1,		CONFIG : 'N U T, 0, 0, 0',
	X = 1222.785  mm,	Y = 98.624  mm,	Z = -238.053  mm,
	W = 0.000 deg,	P = 30.000 deg,	R = 177.979 deg
};
P[74]{
   GP1:
	UF : 0, UT : 1,		CONFIG : 'N U T, 0, 0, 0',
	X = 1222.714  mm,	Y = 96.626  mm,	Z = -238.068  mm,
	W = 0.000 deg,	P = 30.000 deg,	R = 177.979 deg
};
P[75]{
   GP1:
	UF : 0, UT : 1,		CONFIG : 'N U T, 0, 0, 0',
	X = 1222.644  mm,	Y = 94.627  mm,	Z = -238.083  mm,
	W = 0.000 deg,	P = 30.000 deg,	R = -166.376 deg
};
P[76]{
   GP1:
	UF : 0, UT : 1,		CONFIG : 'N U T, 0, 0, 0',
	X = 1222.573  mm,	Y = 92.628  mm,	Z = -238.098  mm,
	W = 0.000 deg,	P = 30.000 deg,	R = -158.394 deg
};
P[77]{
   GP1:
	UF : 0, UT : 1,		CONFIG : 'N U T, 0, 0, 0',
	X = 1222.503  mm,	Y = 90.630  mm,	Z = -238.113  mm,
	W = 0.000 deg,	P = 30.000 deg,	R = -150.412 deg
};
P[78]{
   GP1:
	UF : 0, UT : 1,		CONFIG : 'N U T, 0, 0, 0',
	X = 1222.432  mm,	Y = 88.631  mm,	Z = -238.127  mm,
	W = 0.000 deg,	P = 30.000 deg,	R = -142.430 deg
};
P[79]{
   GP1:
	UF : 0, UT : 1,		CONFIG : 'N U T, 0, 0, 0',
	X = 1222.056  mm,	Y = 89.673  mm,	Z = -238.131  mm,
	W = 0.000 deg,	P = 30.000 deg,	R = -142.111 deg
};
P[80]{
   GP1:
	UF : 0, UT : 1,		CONFIG : 'N U T, 0, 0, 0',
	X = 1217.969  mm,	Y = 85.223  mm,	Z = -238.328  mm,
	W = 0.000 deg,	P = 30.000 deg,	R = -142.111 deg
};
P[81]{
   GP1:
	UF : 0, UT : 1,		CONFIG : 'N U T, 0, 0, 0',
	X = 1219.187  mm,	Y = 83.658  mm,	Z = -238.589  mm,
	W = 0.000 deg,	P = 30.000 deg,	R = -142.111 deg
};
P[82]{
   GP1:
	UF : 0, UT : 1,		CONFIG : 'N U T, 0, 0, 0',
	X = 1220.404  mm,	Y = 82.093  mm,	Z = -238.849  mm,
	W = 0.000 deg,	P = 30.000 deg,	R = -142.111 deg
};
P[83]{
   GP1:
	UF : 0, UT : 1,		CONFIG : 'N U T, 0, 0, 0',
	X = 1226.357  mm,	Y = 84.213  mm,	Z = -239.110  mm,
	W = 0.000 deg,	P = 30.000 deg,	R = -142.111 deg
};
P[84]{
   GP1:
	UF : 0, UT : 1,		CONFIG : 'N U T, 0, 0, 0',
	X = 1222.840  mm,	Y = 78.963  mm,	Z = -239.370  mm,
	W = 0.000 deg,	P = 30.000 deg,	R = -142.111 deg
};
P[85]{
   GP1:
	UF : 0, UT : 1,		CONFIG : 'N U T, 0, 0, 0',
	X = 1224.058  mm,	Y = 77.398  mm,	Z = -239.631  mm,
	W = 0.000 deg,	P = 30.000 deg,	R = -142.111 deg
};
P[86]{
   GP1:
	UF : 0, UT : 1,		CONFIG : 'N U T, 0, 0, 0',
	X = 1230.011  mm,	Y = 79.518  mm,	Z = -239.892  mm,
	W = 0.000 deg,	P = 30.000 deg,	R = -142.111 deg
};
P[87]{
   GP1:
	UF : 0, UT : 1,		CONFIG : 'N U T, 0, 0, 0',
	X = 1226.493  mm,	Y = 74.268  mm,	Z = -240.152  mm,
	W = 0.000 deg,	P = 30.000 deg,	R = -142.111 deg
};
P[88]{
   GP1:
	UF : 0, UT : 1,		CONFIG : 'N U T, 0, 0, 0',
	X = 1227.711  mm,	Y = 72.704  mm,	Z = -240.413  mm,
	W = 0.000 deg,	P = 30.000 deg,	R = -142.111 deg
};
P[89]{
   GP1:
	UF : 0, UT : 1,		CONFIG : 'N U T, 0, 0, 0',
	X = 1233.664  mm,	Y = 74.823  mm,	Z = -240.674  mm,
	W = 0.000 deg,	P = 30.000 deg,	R = -142.111 deg
};
P[90]{
   GP1:
	UF : 0, UT : 1,		CONFIG : 'N U T, 0, 0, 0',
	X = 1234.882  mm,	Y = 73.258  mm,	Z = -240.934  mm,
	W = 0.000 deg,	P = 30.000 deg,	R = -142.111 deg
};
P[91]{
   GP1:
	UF : 0, UT : 1,		CONFIG : 'N U T, 0, 0, 0',
	X = 1231.365  mm,	Y = 68.009  mm,	Z = -241.195  mm,
	W = 0.000 deg,	P = 30.000 deg,	R = -142.111 deg
};
P[92]{
   GP1:
	UF : 0, UT : 1,		CONFIG : 'N U T, 0, 0, 0',
	X = 1232.582  mm,	Y = 66.444  mm,	Z = -241.456  mm,
	W = 0.000 deg,	P = 30.000 deg,	R = -142.111 deg
};
P[93]{
   GP1:
	UF : 0, UT : 1,		CONFIG : 'N U T, 0, 0, 0',
	X = 1238.535  mm,	Y = 68.564  mm,	Z = -241.716  mm,
	W = 0.000 deg,	P = 30.000 deg,	R = -142.111 deg
};
P[94]{
   GP1:
	UF : 0, UT : 1,		CONFIG : 'N U T, 0, 0, 0',
	X = 1235.018  mm,	Y = 63.314  mm,	Z = -241.977  mm,
	W = 0.000 deg,	P = 30.000 deg,	R = -142.111 deg
};
P[95]{
   GP1:
	UF : 0, UT : 1,		CONFIG : 'N U T, 0, 0, 0',
	X = 1236.236  mm,	Y = 61.749  mm,	Z = -242.237  mm,
	W = 0.000 deg,	P = 30.000 deg,	R = -142.111 deg
};
P[96]{
   GP1:
	UF : 0, UT : 1,		CONFIG : 'N U T, 0, 0, 0',
	X = 1242.189  mm,	Y = 63.869  mm,	Z = -242.498  mm,
	W = 0.000 deg,	P = 30.000 deg,	R = -142.111 deg
};
P[97]{
   GP1:
	UF : 0, UT : 1,		CONFIG : 'N U T, 0, 0, 0',
	X = 1238.671  mm,	Y = 58.619  mm,	Z = -242.759  mm,
	W = 0.000 deg,	P = 30.000 deg,	R = -142.111 deg
};
P[98]{
   GP1:
	UF : 0, UT : 1,		CONFIG : 'N U T, 0, 0, 0',
	X = 1239.889  mm,	Y = 57.054  mm,	Z = -243.019  mm,
	W = 0.000 deg,	P = 30.000 deg,	R = -142.111 deg
};
P[99]{
   GP1:
	UF : 0, UT : 1,		CONFIG : 'N U T, 0, 0, 0',
	X = 1245.842  mm,	Y = 59.174  mm,	Z = -243.280  mm,
	W = 0.000 deg,	P = 30.000 deg,	R = -142.111 deg
};
P[100]{
   GP1:
	UF : 0, UT : 1,		CONFIG : 'N U T, 0, 0, 0',
	X = 1242.325  mm,	Y = 53.924  mm,	Z = -243.541  mm,
	W = 0.000 deg,	P = 30.000 deg,	R = -142.111 deg
};
P[101]{
   GP1:
	UF : 0, UT : 1,		CONFIG : 'N U T, 0, 0, 0',
	X = 1243.542  mm,	Y = 52.359  mm,	Z = -243.801  mm,
	W = 0.000 deg,	P = 30.000 deg,	R = -142.111 deg
};
P[102]{
   GP1:
	UF : 0, UT : 1,		CONFIG : 'N U T, 0, 0, 0',
	X = 1244.760  mm,	Y = 50.794  mm,	Z = -244.062  mm,
	W = 0.000 deg,	P = 30.000 deg,	R = -147.811 deg
};
P[103]{
   GP1:
	UF : 0, UT : 1,		CONFIG : 'N U T, 0, 0, 0',
	X = 1245.978  mm,	Y = 49.229  mm,	Z = -244.323  mm,
	W = 0.000 deg,	P = 30.000 deg,	R = -155.358 deg
};
P[104]{
   GP1:
	UF : 0, UT : 1,		CONFIG : 'N U T, 0, 0, 0',
	X = 1247.196  mm,	Y = 47.664  mm,	Z = -244.583  mm,
	W = 0.000 deg,	P = 30.000 deg,	R = -162.905 deg
};
P[105]{
   GP1:
	UF : 0, UT : 1,		CONFIG : 'N U T, 0, 0, 0',
	X = 1248.413  mm,	Y = 46.099  mm,	Z = -244.844  mm,
	W = 0.000 deg,	P = 30.000 deg,	R = -170.452 deg
};
P[106]{
   GP1:
	UF : 0, UT : 1,		CONFIG : 'N U T, 0, 0, 0',
	X = 1249.631  mm,	Y = 44.534  mm,	Z = -245.104  mm,
	W = 0.000 deg,	P = 30.000 deg,	R = -177.999 deg
};
P[107]{
   GP1:
	UF : 0, UT : 1,		CONFIG : 'N U T, 0, 0, 0',
	X = 1250.849  mm,	Y = 42.969  mm,	Z = -245.365  mm,
	W = 0.000 deg,	P = 30.000 deg,	R = -179.846 deg
};
P[108]{
   GP1:
	UF : 0, UT : 1,		CONFIG : 'N U T, 0, 0, 0',
	X = 1250.438  mm,	Y = 44.227  mm,	Z = -245.409  mm,
	W = 0.000 deg,	P = 30.000 deg,	R = -179.846 deg
};
P[109]{
   GP1:
	UF : 0, UT : 1,		CONFIG : 'N U T, 0, 0, 0',
	X = 1250.425  mm,	Y = 42.877  mm,	Z = -245.431  mm,
	W = 0.000 deg,	P = 30.000 deg,	R = -179.846 deg
};
P[110]{
   GP1:
	UF : 0, UT : 1,		CONFIG : 'N U T, 0, 0, 0',
	X = 1250.431  mm,	Y = 40.877  mm,	Z = -245.457  mm,
	W = 0.000 deg,	P = 30.000 deg,	R = -179.846 deg
};
P[111]{
   GP1:
	UF : 0, UT : 1,		CONFIG : 'N U T, 0, 0, 0',
	X = 1250.436  mm,	Y = 38.877  mm,	Z = -245.483  mm,
	W = 0.000 deg,	P = 30.000 deg,	R = -179.846 deg
};
P[112]{
   GP1:
	UF : 0, UT : 1,		CONFIG : 'N U T, 0, 0, 0',
	X = 1250.441  mm,	Y = 36.877  mm,	Z = -245.510  mm,
	W = 0.000 deg,	P = 30.000 deg,	R = -179.846 deg
};
P[113]{
   GP1:
	UF : 0, UT : 1,		CONFIG : 'N U T, 0, 0, 0',
	X = 1250.447  mm,	Y = 34.878  mm,	Z = -245.536  mm,
	W = 0.000 deg,	P = 30.000 deg,	R = -179.846 deg
};
P[114]{
   GP1:
	UF : 0, UT : 1,		CONFIG : 'N U T, 0, 0, 0',
	X = 1256.452  mm,	Y = 32.894  mm,	Z = -245.562  mm,
	W = 0.000 deg,	P = 30.000 deg,	R = -179.846 deg
};
P[115]{
   GP1:
	UF : 0, UT : 1,		CONFIG : 'N U T, 0, 0, 0',
	X = 1256.457  mm,	Y = 30.894  mm,	Z = -245.589  mm,
	W = 0.000 deg,	P = 30.000 deg,	R = -179.846 deg
};
P[116]{
   GP1:
	UF : 0, UT : 1,		CONFIG : 'N U T, 0, 0, 0',
	X = 1250.463  mm,	Y = 28.878  mm,	Z = -245.615  mm,
	W = 0.000 deg,	P = 30.000 deg,	R = -179.846 deg
};
P[117]{
   GP1:
	UF : 0, UT : 1,		CONFIG : 'N U T, 0, 0, 0',
	X = 1250.468  mm,	Y = 26.878  mm,	Z = -245.641  mm,
	W = 0.000 deg,	P = 30.000 deg,	R = -179.846 deg
};
P[118]{
   GP1:
	UF : 0, UT : 1,		CONFIG : 'N U T, 0, 0, 0',
	X = 1250.473  mm,	Y = 24.878  mm,	Z = -245.668  mm,
	W = 0.000 deg,	P = 30.000 deg,	R = -179.846 deg
};
P[119]{
   GP1:
	UF : 0, UT : 1,		CONFIG : 'N U T, 0, 0, 0',
	X = 1250.479  mm,	Y = 22.879  mm,	Z = -245.694  mm,
	W = 0.000 deg,	P = 30.000 deg,	R = -179.846 deg
};
P[120]{
   GP1:
	UF : 0, UT : 1,		CONFIG : 'N U T, 0, 0, 0',
	X = 1250.484  mm,	Y = 20.879  mm,	Z = -245.720  mm,
	W = 0.000 deg,	P = 30.000 deg,	R = -179.846 deg
};
P[121]{
   GP1:
	UF : 0, UT : 1,		CONFIG : 'N U T, 0, 0, 0',
	X = 1250.489  mm,	Y = 18.879  mm,	Z = -245.747  mm,
	W = 0.000 deg,	P = 30.000 deg,	R = -179.846 deg
};
P[122]{
   GP1:
	UF : 0, UT : 1,		CONFIG : 'N U T, 0, 0, 0',
	X = 1250.495  mm,	Y = 16.879  mm,	Z = -245.773  mm,
	W = 0.000 deg,	P = 30.000 deg,	R = -179.846 deg
};
P[123]{
   GP1:
	UF : 0, UT : 1,		CONFIG : 'N U T, 0, 0, 0',
	X = 1250.500  mm,	Y = 14.879  mm,	Z = -245.799  mm,
	W = 0.000 deg,	P = 30.000 deg,	R = -179.846 deg
};
P[124]{
   GP1:
	UF : 0, UT : 1,		CONFIG : 'N U T, 0, 0, 0',
	X = 1250.506  mm,	Y = 12.880  mm,	Z = -245.826  mm,
	W = 0.000 deg,	P = 30.000 deg,	R = -179.846 deg
};
P[125]{
   GP1:
	UF : 0, UT : 1,		CONFIG : 'N U T, 0, 0, 0',
	X = 1250.511  mm,	Y = 10.880  mm,	Z = -245.852  mm,
	W = 0.000 deg,	P = 30.000 deg,	R = -179.846 deg
};
P[126]{
   GP1:
	UF : 0, UT : 1,		CONFIG : 'N U T, 0, 0, 0',
	X = 1250.516  mm,	Y = 8.880  mm,	Z = -245.878  mm,
	W = 0.000 deg,	P = 30.000 deg,	R = -179.846 deg
};
P[127]{
   GP1:
	UF : 0, UT : 1,		CONFIG : 'N U T, 0, 0, 0',
	X = 1250.522  mm,	Y = 6.880  mm,	Z = -245.905  mm,
	W = 0.000 deg,	P = 30.000 deg,	R = -179.846 deg
};
P[128]{
   GP1:
	UF : 0, UT : 1,		CONFIG : 'N U T, 0, 0, 0',
	X = 1250.527  mm,	Y = 4.880  mm,	Z = -245.931  mm,
	W = 0.000 deg,	P = 30.000 deg,	R = -179.846 deg
};
P[129]{
   GP1:
	UF : 0, UT : 1,		CONFIG : 'N U T, 0, 0, 0',
	X = 1250.532  mm,	Y = 2.880  mm,	Z = -245.958  mm,
	W = 0.000 deg,	P = 30.000 deg,	R = -179.846 deg
};
P[130]{
   GP1:
	UF : 0, UT : 1,		CONFIG : 'N U T, 0, 0, 0',
	X = 1250.538  mm,	Y = 0.881  mm,	Z = -245.984  mm,
	W = 0.000 deg,	P = 30.000 deg,	R = -179.846 deg
};
P[131]{
   GP1:
	UF : 0, UT : 1,		CONFIG : 'N U T, 0, 0, 0',
	X = 1250.543  mm,	Y = -1.119  mm,	Z = -246.010  mm,
	W = 0.000 deg,	P = 30.000 deg,	R = -179.846 deg
};
P[132]{
   GP1:
	UF : 0, UT : 1,		CONFIG : 'N U T, 0, 0, 0',
	X = 1250.548  mm,	Y = -3.119  mm,	Z = -246.037  mm,
	W = 0.000 deg,	P = 30.000 deg,	R = -179.846 deg
};
P[133]{
   GP1:
	UF : 0, UT : 1,		CONFIG : 'N U T, 0, 0, 0',
	X = 1250.554  mm,	Y = -5.119  mm,	Z = -246.063  mm,
	W = 0.000 deg,	P = 30.000 deg,	R = -179.846 deg
};
P[134]{
   GP1:
	UF : 0, UT : 1,		CONFIG : 'N U T, 0, 0, 0',
	X = 1250.559  mm,	Y = -7.119  mm,	Z = -246.089  mm,
	W = 0.000 deg,	P = 30.000 deg,	R = -179.846 deg
};
P[135]{
   GP1:
	UF : 0, UT : 1,		CONFIG : 'N U T, 0, 0, 0',
	X = 1250.565  mm,	Y = -9.118  mm,	Z = -246.116  mm,
	W = 0.000 deg,	P = 30.000 deg,	R = -179.846 deg
};
P[136]{
   GP1:
	UF : 0, UT : 1,		CONFIG : 'N U T, 0, 0, 0',
	X = 1256.570  mm,	Y = -11.102  mm,	Z = -246.142  mm,
	W = 0.000 deg,	P = 30.000 deg,	R = -179.846 deg
};
P[137]{
   GP1:
	UF : 0, UT : 1,		CONFIG : 'N U T, 0, 0, 0',
	X = 1256.575  mm,	Y = -13.102  mm,	Z = -246.168  mm,
	W = 0.000 deg,	P = 30.000 deg,	R = -179.846 deg
};
P[138]{
   GP1:
	UF : 0, UT : 1,		CONFIG : 'N U T, 0, 0, 0',
	X = 1250.581  mm,	Y = -15.118  mm,	Z = -246.195  mm,
	W = 0.000 deg,	P = 30.000 deg,	R = 173.432 deg
};
P[139]{
   GP1:
	UF : 0, UT : 1,		CONFIG : 'N U T, 0, 0, 0',
	X = 1250.586  mm,	Y = -17.118  mm,	Z = -246.221  mm,
	W = 0.000 deg,	P = 30.000 deg,	R = 165.358 deg
};
P[140]{
   GP1:
	UF : 0, UT : 1,		CONFIG : 'N U T, 0, 0, 0',
	X = 1250.591  mm,	Y = -19.118  mm,	Z = -246.247  mm,
	W = 0.000 deg,	P = 30.000 deg,	R = 157.284 deg
};
P[141]{
   GP1:
	UF : 0, UT : 1,		CONFIG : 'N U T, 0, 0, 0',
	X = 1250.597  mm,	Y = -21.117  mm,	Z = -246.274  mm,
	W = 0.000 deg,	P = 30.000 deg,	R = 149.209 deg
};
P[142]{
   GP1:
	UF : 0, UT : 1,		CONFIG : 'N U T, 0, 0, 0',
	X = 1250.602  mm,	Y = -23.117  mm,	Z = -246.300  mm,
	W = 0.000 deg,	P = 30.000 deg,	R = 141.135 deg
};
P[143]{
   GP1:
	UF : 0, UT : 1,		CONFIG : 'N U T, 0, 0, 0',
	X = 1250.613  mm,	Y = -24.725  mm,	Z = -246.324  mm,
	W = 0.000 deg,	P = 30.000 deg,	R = 139.782 deg
};
P[144]{
   GP1:
	UF : 0, UT : 1,		CONFIG : 'N U T, 0, 0, 0',
	X = 1251.190  mm,	Y = -23.124  mm,	Z = -246.300  mm,
	W = 0.000 deg,	P = 30.000 deg,	R = 139.782 deg
};
P[145]{
   GP1:
	UF : 0, UT : 1,		CONFIG : 'N U T, 0, 0, 0',
	X = 1249.908  mm,	Y = -24.640  mm,	Z = -246.055  mm,
	W = 0.000 deg,	P = 30.000 deg,	R = 139.782 deg
};
P[146]{
   GP1:
	UF : 0, UT : 1,		CONFIG : 'N U T, 0, 0, 0',
	X = 1248.626  mm,	Y = -26.156  mm,	Z = -245.811  mm,
	W = 0.000 deg,	P = 30.000 deg,	R = 139.782 deg
};
P[147]{
   GP1:
	UF : 0, UT : 1,		CONFIG : 'N U T, 0, 0, 0',
	X = 1251.926  mm,	Y = -31.546  mm,	Z = -245.567  mm,
	W = 0.000 deg,	P = 30.000 deg,	R = 139.782 deg
};
P[148]{
   GP1:
	UF : 0, UT : 1,		CONFIG : 'N U T, 0, 0, 0',
	X = 1246.063  mm,	Y = -29.187  mm,	Z = -245.323  mm,
	W = 0.000 deg,	P = 30.000 deg,	R = 139.782 deg
};
P[149]{
   GP1:
	UF : 0, UT : 1,		CONFIG : 'N U T, 0, 0, 0',
	X = 1244.781  mm,	Y = -30.703  mm,	Z = -245.079  mm,
	W = 0.000 deg,	P = 30.000 deg,	R = 139.782 deg
};
P[150]{
   GP1:
	UF : 0, UT : 1,		CONFIG : 'N U T, 0, 0, 0',
	X = 1248.081  mm,	Y = -36.093  mm,	Z = -244.835  mm,
	W = 0.000 deg,	P = 30.000 deg,	R = 139.782 deg
};
P[151]{
   GP1:
	UF : 0, UT : 1,		CONFIG : 'N U T, 0, 0, 0',
	X = 1242.217  mm,	Y = -33.735  mm,	Z = -244.590  mm,
	W = 0.000 deg,	P = 30.000 deg,	R = 139.782 deg
};
P[152]{
   GP1:
	UF : 0, UT : 1,		CONFIG : 'N U T, 0, 0, 0',
	X = 1240.936  mm,	Y = -35.250  mm,	Z = -244.346  mm,
	W = 0.000 deg,	P = 30.000 deg,	R = 139.782 deg
};
P[153]{
   GP1:
	UF : 0, UT : 1,		CONFIG : 'N U T, 0, 0, 0',
	X = 1239.654  mm,	Y = -36.766  mm,	Z = -244.102  mm,
	W = 0.000 deg,	P = 30.000 deg,	R = 139.782 deg
};
P[154]{
   GP1:
	UF : 0, UT : 1,		CONFIG : 'N U T, 0, 0, 0',
	X = 1238.372  mm,	Y = -38.282  mm,	Z = -243.858  mm,
	W = 0.000 deg,	P = 30.000 deg,	R = 139.782 deg
};
P[155]{
   GP1:
	UF : 0, UT : 1,		CONFIG : 'N U T, 0, 0, 0',
	X = 1241.672  mm,	Y = -43.672  mm,	Z = -243.614  mm,
	W = 0.000 deg,	P = 30.000 deg,	R = 139.782 deg
};
P[156]{
   GP1:
	UF : 0, UT : 1,		CONFIG : 'N U T, 0, 0, 0',
	X = 1235.809  mm,	Y = -41.313  mm,	Z = -243.370  mm,
	W = 0.000 deg,	P = 30.000 deg,	R = 139.782 deg
};
P[157]{
   GP1:
	UF : 0, UT : 1,		CONFIG : 'N U T, 0, 0, 0',
	X = 1234.527  mm,	Y = -42.829  mm,	Z = -243.126  mm,
	W = 0.000 deg,	P = 30.000 deg,	R = 139.782 deg
};
P[158]{
   GP1:
	UF : 0, UT : 1,		CONFIG : 'N U T, 0, 0, 0',
	X = 1237.827  mm,	Y = -48.219  mm,	Z = -242.881  mm,
	W = 0.000 deg,	P = 30.000 deg,	R = 139.782 deg
};
P[159]{
   GP1:
	UF : 0, UT : 1,		CONFIG : 'N U T, 0, 0, 0',
	X = 1231.964  mm,	Y = -45.861  mm,	Z = -242.637  mm,
	W = 0.000 deg,	P = 30.000 deg,	R = 139.782 deg
};
P[160]{
   GP1:
	UF : 0, UT : 1,		CONFIG : 'N U T, 0, 0, 0',
	X = 1230.682  mm,	Y = -47.376  mm,	Z = -242.393  mm,
	W = 0.000 deg,	P = 30.000 deg,	R = 139.782 deg
};
P[161]{
   GP1:
	UF : 0, UT : 1,		CONFIG : 'N U T, 0, 0, 0',
	X = 1229.400  mm,	Y = -48.892  mm,	Z = -242.149  mm,
	W = 0.000 deg,	P = 30.000 deg,	R = 139.782 deg
};
P[162]{
   GP1:
	UF : 0, UT : 1,		CONFIG : 'N U T, 0, 0, 0',
	X = 1228.118  mm,	Y = -50.408  mm,	Z = -241.905  mm,
	W = 0.000 deg,	P = 30.000 deg,	R = 139.782 deg
};
P[163]{
   GP1:
	UF : 0, UT : 1,		CONFIG : 'N U T, 0, 0, 0',
	X = 1231.418  mm,	Y = -55.798  mm,	Z = -241.661  mm,
	W = 0.000 deg,	P = 30.000 deg,	R = 139.782 deg
};
P[164]{
   GP1:
	UF : 0, UT : 1,		CONFIG : 'N U T, 0, 0, 0',
	X = 1225.555  mm,	Y = -53.440  mm,	Z = -241.416  mm,
	W = 0.000 deg,	P = 30.000 deg,	R = 139.782 deg
};
P[165]{
   GP1:
	UF : 0, UT : 1,		CONFIG : 'N U T, 0, 0, 0',
	X = 1224.273  mm,	Y = -54.955  mm,	Z = -241.172  mm,
	W = 0.000 deg,	P = 30.000 deg,	R = 139.782 deg
};
P[166]{
   GP1:
	UF : 0, UT : 1,		CONFIG : 'N U T, 0, 0, 0',
	X = 1227.573  mm,	Y = -60.345  mm,	Z = -240.928  mm,
	W = 0.000 deg,	P = 30.000 deg,	R = 140.523 deg
};
P[167]{
   GP1:
	UF : 0, UT : 1,		CONFIG : 'N U T, 0, 0, 0',
	X = 1226.291  mm,	Y = -61.861  mm,	Z = -240.684  mm,
	W = 0.000 deg,	P = 30.000 deg,	R = 148.024 deg
};
P[168]{
   GP1:
	UF : 0, UT : 1,		CONFIG : 'N U T, 0, 0, 0',
	X = 1225.010  mm,	Y = -63.377  mm,	Z = -240.440  mm,
	W = 0.000 deg,	P = 30.000 deg,	R = 155.526 deg
};
P[169]{
   GP1:
	UF : 0, UT : 1,		CONFIG : 'N U T, 0, 0, 0',
	X = 1223.728  mm,	Y = -64.893  mm,	Z = -240.196  mm,
	W = 0.000 deg,	P = 30.000 deg,	R = 163.028 deg
};
P[170]{
   GP1:
	UF : 0, UT : 1,		CONFIG : 'N U T, 0, 0, 0',
	X = 1222.446  mm,	Y = -66.408  mm,	Z = -239.952  mm,
	W = 0.000 deg,	P = 30.000 deg,	R = 170.530 deg
};
P[171]{
   GP1:
	UF : 0, UT : 1,		CONFIG : 'N U T, 0, 0, 0',
	X = 1221.165  mm,	Y = -67.924  mm,	Z = -239.707  mm,
	W = 0.000 deg,	P = 30.000 deg,	R = 177.291 deg
};
P[172]{
   GP1:
	UF : 0, UT : 1,		CONFIG : 'N U T, 0, 0, 0',
	X = 1221.665  mm,	Y = -66.607  mm,	Z = -239.673  mm,
	W = 0.000 deg,	P = 30.000 deg,	R = 177.291 deg
};
P[173]{
   GP1:
	UF : 0, UT : 1,		CONFIG : 'N U T, 0, 0, 0',
	X = 1221.608  mm,	Y = -68.058  mm,	Z = -239.686  mm,
	W = 0.000 deg,	P = 30.000 deg,	R = 177.291 deg
};
P[174]{
   GP1:
	UF : 0, UT : 1,		CONFIG : 'N U T, 0, 0, 0',
	X = 1221.513  mm,	Y = -70.056  mm,	Z = -239.702  mm,
	W = 0.000 deg,	P = 30.000 deg,	R = 177.291 deg
};
P[175]{
   GP1:
	UF : 0, UT : 1,		CONFIG : 'N U T, 0, 0, 0',
	X = 1215.425  mm,	Y = -71.770  mm,	Z = -239.717  mm,
	W = 0.000 deg,	P = 30.000 deg,	R = 177.291 deg
};
P[176]{
   GP1:
	UF : 0, UT : 1,		CONFIG : 'N U T, 0, 0, 0',
	X = 1221.324  mm,	Y = -74.051  mm,	Z = -239.733  mm,
	W = 0.000 deg,	P = 30.000 deg,	R = 177.291 deg
};
P[177]{
   GP1:
	UF : 0, UT : 1,		CONFIG : 'N U T, 0, 0, 0',
	X = 1221.230  mm,	Y = -76.049  mm,	Z = -239.748  mm,
	W = 0.000 deg,	P = 30.000 deg,	R = 177.291 deg
};
P[178]{
   GP1:
	UF : 0, UT : 1,		CONFIG : 'N U T, 0, 0, 0',
	X = 1215.142  mm,	Y = -77.763  mm,	Z = -239.764  mm,
	W = 0.000 deg,	P = 30.000 deg,	R = 177.291 deg
};
P[179]{
   GP1:
	UF : 0, UT : 1,		CONFIG : 'N U T, 0, 0, 0',
	X = 1221.040  mm,	Y = -80.044  mm,	Z = -239.780  mm,
	W = 0.000 deg,	P = 30.000 deg,	R = 177.291 deg
};
P[180]{
   GP1:
	UF : 0, UT : 1,		CONFIG : 'N U T, 0, 0, 0',
	X = 1220.946  mm,	Y = -82.042  mm,	Z = -239.795  mm,
	W = 0.000 deg,	P = 30.000 deg,	R = 177.291 deg
};
P[181]{
   GP1:
	UF : 0, UT : 1,		CONFIG : 'N U T, 0, 0, 0',
	X = 1220.851  mm,	Y = -84.040  mm,	Z = -239.811  mm,
	W = 0.000 deg,	P = 30.000 deg,	R = 177.291 deg
};
P[182]{
   GP1:
	UF : 0, UT : 1,		CONFIG : 'N U T, 0, 0, 0',
	X = 1220.757  mm,	Y = -86.038  mm,	Z = -239.826  mm,
	W = 0.000 deg,	P = 30.000 deg,	R = 177.291 deg
};
P[183]{
   GP1:
	UF : 0, UT : 1,		CONFIG : 'N U T, 0, 0, 0',
	X = 1214.669  mm,	Y = -87.752  mm,	Z = -239.842  mm,
	W = 0.000 deg,	P = 30.000 deg,	R = 177.291 deg
};
P[184]{
   GP1:
	UF : 0, UT : 1,		CONFIG : 'N U T, 0, 0, 0',
	X = 1220.568  mm,	Y = -90.033  mm,	Z = -239.857  mm,
	W = 0.000 deg,	P = 30.000 deg,	R = 177.291 deg
};
P[185]{
   GP1:
	UF : 0, UT : 1,		CONFIG : 'N U T, 0, 0, 0',
	X = 1220.473  mm,	Y = -92.031  mm,	Z = -239.873  mm,
	W = 0.000 deg,	P = 30.000 deg,	R = 177.291 deg
};
P[186]{
   GP1:
	UF : 0, UT : 1,		CONFIG : 'N U T, 0, 0, 0',
	X = 1214.386  mm,	Y = -93.745  mm,	Z = -239.888  mm,
	W = 0.000 deg,	P = 30.000 deg,	R = 177.291 deg
};
P[187]{
   GP1:
	UF : 0, UT : 1,		CONFIG : 'N U T, 0, 0, 0',
	X = 1220.284  mm,	Y = -96.026  mm,	Z = -239.904  mm,
	W = 0.000 deg,	P = 30.000 deg,	R = 177.291 deg
};
P[188]{
   GP1:
	UF : 0, UT : 1,		CONFIG : 'N U T, 0, 0, 0',
	X = 1220.190  mm,	Y = -98.024  mm,	Z = -239.920  mm,
	W = 0.000 deg,	P = 30.000 deg,	R = 177.291 deg
};
P[189]{
   GP1:
	UF : 0, UT : 1,		CONFIG : 'N U T, 0, 0, 0',
	X = 1214.102  mm,	Y = -99.738  mm,	Z = -239.935  mm,
	W = 0.000 deg,	P = 30.000 deg,	R = 177.291 deg
};
P[190]{
   GP1:
	UF : 0, UT : 1,		CONFIG : 'N U T, 0, 0, 0',
	X = 1220.001  mm,	Y = -102.019  mm,	Z = -239.951  mm,
	W = 0.000 deg,	P = 30.000 deg,	R = 177.291 deg
};
P[191]{
   GP1:
	UF : 0, UT : 1,		CONFIG : 'N U T, 0, 0, 0',
	X = 1219.906  mm,	Y = -104.017  mm,	Z = -239.966  mm,
	W = 0.000 deg,	P = 30.000 deg,	R = 177.291 deg
};
P[192]{
   GP1:
	UF : 0, UT : 1,		CONFIG : 'N U T, 0, 0, 0',
	X = 1219.812  mm,	Y = -106.015  mm,	Z = -239.982  mm,
	W = 0.000 deg,	P = 30.000 deg,	R = 177.291 deg
};
P[193]{
   GP1:
	UF : 0, UT : 1,		CONFIG : 'N U T, 0, 0, 0',
	X = 1219.717  mm,	Y = -108.012  mm,	Z = -239.997  mm,
	W = 0.000 deg,	P = 30.000 deg,	R = 177.291 deg
};
P[194]{
   GP1:
	UF : 0, UT : 1,		CONFIG : 'N U T, 0, 0, 0',
	X = 1213.629  mm,	Y = -109.726  mm,	Z = -240.013  mm,
	W = 0.000 deg,	P = 30.000 deg,	R = 177.291 deg
};
P[195]{
   GP1:
	UF : 0, UT : 1,		CONFIG : 'N U T, 0, 0, 0',
	X = 1219.528  mm,	Y = -112.008  mm,	Z = -240.029  mm,
	W = 0.000 deg,	P = 30.000 deg,	R = 177.291 deg
};
P[196]{
   GP1:
	UF : 0, UT : 1,		CONFIG : 'N U T, 0, 0, 0',
	X = 1219.434  mm,	Y = -114.005  mm,	Z = -240.044  mm,
	W = 0.000 deg,	P = 30.000 deg,	R = 177.291 deg
};
P[197]{
   GP1:
	UF : 0, UT : 1,		CONFIG : 'N U T, 0, 0, 0',
	X = 1213.346  mm,	Y = -115.720  mm,	Z = -240.060  mm,
	W = 0.000 deg,	P = 30.000 deg,	R = 177.291 deg
};
P[198]{
   GP1:
	UF : 0, UT : 1,		CONFIG : 'N U T, 0, 0, 0',
	X = 1219.245  mm,	Y = -118.001  mm,	Z = -240.075  mm,
	W = 0.000 deg,	P = 30.000 deg,	R = 177.291 deg
};
P[199]{
   GP1:
	UF : 0, UT : 1,		CONFIG : 'N U T, 0, 0, 0',
	X = 1219.150  mm,	Y = -119.999  mm,	Z = -240.091  mm,
	W = 0.000 deg,	P = 30.000 deg,	R = 177.291 deg
};
P[200]{
   GP1:
	UF : 0, UT : 1,		CONFIG : 'N U T, 0, 0, 0',
	X = 1213.062  mm,	Y = -121.713  mm,	Z = -240.106  mm,
	W = 0.000 deg,	P = 30.000 deg,	R = 177.291 deg
};
P[201]{
   GP1:
	UF : 0, UT : 1,		CONFIG : 'N U T, 0, 0, 0',
	X = 1218.961  mm,	Y = -123.994  mm,	Z = -240.122  mm,
	W = 0.000 deg,	P = 30.000 deg,	R = 177.291 deg
};
P[202]{
   GP1:
	UF : 0, UT : 1,		CONFIG : 'N U T, 0, 0, 0',
	X = 1218.866  mm,	Y = -125.992  mm,	Z = -240.138  mm,
	W = 0.000 deg,	P = 30.000 deg,	R = 177.291 deg
};
P[203]{
   GP1:
	UF : 0, UT : 1,		CONFIG : 'N U T, 0, 0, 0',
	X = 1218.772  mm,	Y = -127.989  mm,	Z = -240.153  mm,
	W = 0.000 deg,	P = 30.000 deg,	R = -175.883 deg
};
P[204]{
   GP1:
	UF : 0, UT : 1,		CONFIG : 'N U T, 0, 0, 0',
	X = 1218.677  mm,	Y = -129.987  mm,	Z = -240.169  mm,
	W = 0.000 deg,	P = 30.000 deg,	R = -167.929 deg
};
P[205]{
   GP1:
	UF : 0, UT : 1,		CONFIG : 'N U T, 0, 0, 0',
	X = 1218.583  mm,	Y = -131.985  mm,	Z = -240.184  mm,
	W = 0.000 deg,	P = 30.000 deg,	R = -159.976 deg
};
P[206]{
   GP1:
	UF : 0, UT : 1,		CONFIG : 'N U T, 0, 0, 0',
	X = 1218.488  mm,	Y = -133.982  mm,	Z = -240.200  mm,
	W = 0.000 deg,	P = 30.000 deg,	R = -152.023 deg
};
P[207]{
   GP1:
	UF : 0, UT : 1,		CONFIG : 'N U T, 0, 0, 0',
	X = 1218.394  mm,	Y = -135.980  mm,	Z = -240.215  mm,
	W = 0.000 deg,	P = 30.000 deg,	R = -144.069 deg
};
P[208]{
   GP1:
	UF : 0, UT : 1,		CONFIG : 'N U T, 0, 0, 0',
	X = 1217.963  mm,	Y = -134.648  mm,	Z = -240.218  mm,
	W = 0.000 deg,	P = 30.000 deg,	R = -142.942 deg
};
P[209]{
   GP1:
	UF : 0, UT : 1,		CONFIG : 'N U T, 0, 0, 0',
	X = 1213.981  mm,	Y = -139.300  mm,	Z = -240.421  mm,
	W = 0.000 deg,	P = 30.000 deg,	R = -142.942 deg
};
P[210]{
   GP1:
	UF : 0, UT : 1,		CONFIG : 'N U T, 0, 0, 0',
	X = 1215.178  mm,	Y = -140.884  mm,	Z = -240.666  mm,
	W = 0.000 deg,	P = 30.000 deg,	R = -142.942 deg
};
P[211]{
   GP1:
	UF : 0, UT : 1,		CONFIG : 'N U T, 0, 0, 0',
	X = 1221.162  mm,	Y = -138.853  mm,	Z = -240.911  mm,
	W = 0.000 deg,	P = 30.000 deg,	R = -142.942 deg
};
P[212]{
   GP1:
	UF : 0, UT : 1,		CONFIG : 'N U T, 0, 0, 0',
	X = 1222.358  mm,	Y = -140.437  mm,	Z = -241.156  mm,
	W = 0.000 deg,	P = 30.000 deg,	R = -142.942 deg
};
P[213]{
   GP1:
	UF : 0, UT : 1,		CONFIG : 'N U T, 0, 0, 0',
	X = 1223.554  mm,	Y = -142.021  mm,	Z = -241.401  mm,
	W = 0.000 deg,	P = 30.000 deg,	R = -142.942 deg
};
P[214]{
   GP1:
	UF : 0, UT : 1,		CONFIG : 'N U T, 0, 0, 0',
	X = 1224.750  mm,	Y = -143.605  mm,	Z = -241.645  mm,
	W = 0.000 deg,	P = 30.000 deg,	R = -142.942 deg
};
P[215]{
   GP1:
	UF : 0, UT : 1,		CONFIG : 'N U T, 0, 0, 0',
	X = 1225.947  mm,	Y = -145.189  mm,	Z = -241.890  mm,
	W = 0.000 deg,	P = 30.000 deg,	R = -142.942 deg
};
P[216]{
   GP1:
	UF : 0, UT : 1,		CONFIG : 'N U T, 0, 0, 0',
	X = 1227.143  mm,	Y = -146.773  mm,	Z = -242.135  mm,
	W = 0.000 deg,	P = 30.000 deg,	R = -142.942 deg
};
P[217]{
   GP1:
	UF : 0, UT : 1,		CONFIG : 'N U T, 0, 0, 0',
	X = 1228.339  mm,	Y = -148.357  mm,	Z = -242.380  mm,
	W = 0.000 deg,	P = 30.000 deg,	R = -142.942 deg
};
P[218]{
   GP1:
	UF : 0, UT : 1,		CONFIG : 'N U T, 0, 0, 0',
	X = 1229.535  mm,	Y = -149.941  mm,	Z = -242.624  mm,
	W = 0.000 deg,	P = 30.000 deg,	R = -142.942 deg
};
P[219]{
   GP1:
	UF : 0, UT : 1,		CONFIG : 'N U T, 0, 0, 0',
	X = 1225.943  mm,	Y = -155.141  mm,	Z = -242.869  mm,
	W = 0.000 deg,	P = 30.000 deg,	R = -142.942 deg
};
P[220]{
   GP1:
	UF : 0, UT : 1,		CONFIG : 'N U T, 0, 0, 0',
	X = 1227.139  mm,	Y = -156.725  mm,	Z = -243.114  mm,
	W = 0.000 deg,	P = 30.000 deg,	R = -142.942 deg
};
P[221]{
   GP1:
	UF : 0, UT : 1,		CONFIG : 'N U T, 0, 0, 0',
	X = 1233.124  mm,	Y = -154.693  mm,	Z = -243.359  mm,
	W = 0.000 deg,	P = 30.000 deg,	R = -142.942 deg
};
P[222]{
   GP1:
	UF : 0, UT : 1,		CONFIG : 'N U T, 0, 0, 0',
	X = 1234.320  mm,	Y = -156.277  mm,	Z = -243.604  mm,
	W = 0.000 deg,	P = 30.000 deg,	R = -142.942 deg
};
P[223]{
   GP1:
	UF : 0, UT : 1,		CONFIG : 'N U T, 0, 0, 0',
	X = 1235.516  mm,	Y = -157.861  mm,	Z = -243.848  mm,
	W = 0.000 deg,	P = 30.000 deg,	R = -142.942 deg
};
P[224]{
   GP1:
	UF : 0, UT : 1,		CONFIG : 'N U T, 0, 0, 0',
	X = 1236.712  mm,	Y = -159.445  mm,	Z = -244.093  mm,
	W = 0.000 deg,	P = 30.000 deg,	R = -142.942 deg
};
P[225]{
   GP1:
	UF : 0, UT : 1,		CONFIG : 'N U T, 0, 0, 0',
	X = 1237.908  mm,	Y = -161.029  mm,	Z = -244.338  mm,
	W = 0.000 deg,	P = 30.000 deg,	R = -142.942 deg
};
P[226]{
   GP1:
	UF : 0, UT : 1,		CONFIG : 'N U T, 0, 0, 0',
	X = 1239.105  mm,	Y = -162.614  mm,	Z = -244.583  mm,
	W = 0.000 deg,	P = 30.000 deg,	R = -142.942 deg
};
P[227]{
   GP1:
	UF : 0, UT : 1,		CONFIG : 'N U T, 0, 0, 0',
	X = 1240.301  mm,	Y = -164.198  mm,	Z = -244.827  mm,
	W = 0.000 deg,	P = 30.000 deg,	R = -142.942 deg
};
P[228]{
   GP1:
	UF : 0, UT : 1,		CONFIG : 'N U T, 0, 0, 0',
	X = 1241.497  mm,	Y = -165.782  mm,	Z = -245.072  mm,
	W = 0.000 deg,	P = 30.000 deg,	R = -142.942 deg
};
P[229]{
   GP1:
	UF : 0, UT : 1,		CONFIG : 'N U T, 0, 0, 0',
	X = 1237.905  mm,	Y = -170.981  mm,	Z = -245.317  mm,
	W = 0.000 deg,	P = 30.000 deg,	R = -142.942 deg
};
P[230]{
   GP1:
	UF : 0, UT : 1,		CONFIG : 'N U T, 0, 0, 0',
	X = 1239.101  mm,	Y = -172.565  mm,	Z = -245.562  mm,
	W = 0.000 deg,	P = 30.000 deg,	R = -142.942 deg
};
P[231]{
   GP1:
	UF : 0, UT : 1,		CONFIG : 'N U T, 0, 0, 0',
	X = 1245.085  mm,	Y = -170.534  mm,	Z = -245.806  mm,
	W = 0.000 deg,	P = 30.000 deg,	R = -142.942 deg
};
P[232]{
   GP1:
	UF : 0, UT : 1,		CONFIG : 'N U T, 0, 0, 0',
	X = 1246.282  mm,	Y = -172.118  mm,	Z = -246.051  mm,
	W = 0.000 deg,	P = 30.000 deg,	R = -142.942 deg
};
P[233]{
   GP1:
	UF : 0, UT : 1,		CONFIG : 'N U T, 0, 0, 0',
	X = 1242.690  mm,	Y = -177.318  mm,	Z = -246.296  mm,
	W = 0.000 deg,	P = 30.000 deg,	R = -149.097 deg
};
P[234]{
   GP1:
	UF : 0, UT : 1,		CONFIG : 'N U T, 0, 0, 0',
	X = 1243.886  mm,	Y = -178.902  mm,	Z = -246.541  mm,
	W = 0.000 deg,	P = 30.000 deg,	R = -156.501 deg
};
P[235]{
   GP1:
	UF : 0, UT : 1,		CONFIG : 'N U T, 0, 0, 0',
	X = 1245.082  mm,	Y = -180.486  mm,	Z = -246.786  mm,
	W = 0.000 deg,	P = 30.000 deg,	R = -163.905 deg
};
P[236]{
   GP1:
	UF : 0, UT : 1,		CONFIG : 'N U T, 0, 0, 0',
	X = 1246.278  mm,	Y = -182.070  mm,	Z = -247.030  mm,
	W = 0.000 deg,	P = 30.000 deg,	R = -171.310 deg
};
P[237]{
   GP1:
	UF : 0, UT : 1,		CONFIG : 'N U T, 0, 0, 0',
	X = 1247.474  mm,	Y = -183.654  mm,	Z = -247.275  mm,
	W = 0.000 deg,	P = 30.000 deg,	R = -178.714 deg
};
P[238]{
   GP1:
	UF : 0, UT : 1,		CONFIG : 'N U T, 0, 0, 0',
	X = 1247.122  mm,	Y = -182.515  mm,	Z = -247.323  mm,
	W = 0.000 deg,	P = 30.000 deg,	R = -179.964 deg
};
P[239]{
   GP1:
	UF : 0, UT : 1,		CONFIG : 'N U T, 0, 0, 0',
	X = 1253.101  mm,	Y = -183.763  mm,	Z = -247.354  mm,
	W = 0.000 deg,	P = 30.000 deg,	R = -179.964 deg
};
P[240]{
   GP1:
	UF : 0, UT : 1,		CONFIG : 'N U T, 0, 0, 0',
	X = 1247.103  mm,	Y = -185.767  mm,	Z = -247.392  mm,
	W = 0.000 deg,	P = 30.000 deg,	R = -179.964 deg
};
P[241]{
   GP1:
	UF : 0, UT : 1,		CONFIG : 'N U T, 0, 0, 0',
	X = 1247.104  mm,	Y = -187.766  mm,	Z = -247.430  mm,
	W = 0.000 deg,	P = 30.000 deg,	R = -179.964 deg
};
P[242]{
   GP1:
	UF : 0, UT : 1,		CONFIG : 'N U T, 0, 0, 0',
	X = 1247.105  mm,	Y = -189.766  mm,	Z = -247.469  mm,
	W = 0.000 deg,	P = 30.000 deg,	R = -179.964 deg
};
P[243]{
   GP1:
	UF : 0, UT : 1,		CONFIG : 'N U T, 0, 0, 0',
	X = 1247.106  mm,	Y = -191.766  mm,	Z = -247.507  mm,
	W = 0.000 deg,	P = 30.000 deg,	R = -179.964 deg
};
P[244]{
   GP1:
	UF : 0, UT : 1,		CONFIG : 'N U T, 0, 0, 0',
	X = 1247.108  mm,	Y = -193.765  mm,	Z = -247.545  mm,
	W = 0.000 deg,	P = 30.000 deg,	R = -179.964 deg
};
P[245]{
   GP1:
	UF : 0, UT : 1,		CONFIG : 'N U T, 0, 0, 0',
	X = 1247.109  mm,	Y = -195.765  mm,	Z = -247.584  mm,
	W = 0.000 deg,	P = 30.000 deg,	R = -179.964 deg
};
P[246]{
   GP1:
	UF : 0, UT : 1,		CONFIG : 'N U T, 0, 0, 0',
	X = 1253.110  mm,	Y = -197.761  mm,	Z = -247.622  mm,
	W = 0.000 deg,	P = 30.000 deg,	R = -179.964 deg
};
P[247]{
   GP1:
	UF : 0, UT : 1,		CONFIG : 'N U T, 0, 0, 0',
	X = 1247.111  mm,	Y = -199.764  mm,	Z = -247.660  mm,
	W = 0.000 deg,	P = 30.000 deg,	R = -179.964 deg
};
P[248]{
   GP1:
	UF : 0, UT : 1,		CONFIG : 'N U T, 0, 0, 0',
	X = 1247.113  mm,	Y = -201.764  mm,	Z = -247.699  mm,
	W = 0.000 deg,	P = 30.000 deg,	R = -179.964 deg
};
P[249]{
   GP1:
	UF : 0, UT : 1,		CONFIG : 'N U T, 0, 0, 0',
	X = 1247.114  mm,	Y = -203.763  mm,	Z = -247.737  mm,
	W = 0.000 deg,	P = 30.000 deg,	R = -179.964 deg
};
P[250]{
   GP1:
	UF : 0, UT : 1,		CONFIG : 'N U T, 0, 0, 0',
	X = 1247.115  mm,	Y = -205.763  mm,	Z = -247.775  mm,
	W = 0.000 deg,	P = 30.000 deg,	R = -179.964 deg
};
P[251]{
   GP1:
	UF : 0, UT : 1,		CONFIG : 'N U T, 0, 0, 0',
	X = 1247.116  mm,	Y = -207.763  mm,	Z = -247.814  mm,
	W = 0.000 deg,	P = 30.000 deg,	R = -179.964 deg
};
P[252]{
   GP1:
	UF : 0, UT : 1,		CONFIG : 'N U T, 0, 0, 0',
	X = 1247.118  mm,	Y = -209.762  mm,	Z = -247.852  mm,
	W = 0.000 deg,	P = 30.000 deg,	R = -179.964 deg
};
P[253]{
   GP1:
	UF : 0, UT : 1,		CONFIG : 'N U T, 0, 0, 0',
	X = 1247.119  mm,	Y = -211.762  mm,	Z = -247.890  mm,
	W = 0.000 deg,	P = 30.000 deg,	R = -179.964 deg
};
P[254]{
   GP1:
	UF : 0, UT : 1,		CONFIG : 'N U T, 0, 0, 0',
	X = 1247.120  mm,	Y = -213.761  mm,	Z = -247.929  mm,
	W = 0.000 deg,	P = 30.000 deg,	R = -179.964 deg
};
P[255]{
   GP1:
	UF : 0, UT : 1,		CONFIG : 'N U T, 0, 0, 0',
	X = 1253.121  mm,	Y = -215.757  mm,	Z = -247.967  mm,
	W = 0.000 deg,	P = 30.000 deg,	R = -179.964 deg
};
P[256]{
   GP1:
	UF : 0, UT : 1,		CONFIG : 'N U T, 0, 0, 0',
	X = 1247.123  mm,	Y = -217.761  mm,	Z = -248.005  mm,
	W = 0.000 deg,	P = 30.000 deg,	R = -179.964 deg
};
P[257]{
   GP1:
	UF : 0, UT : 1,		CONFIG : 'N U T, 0, 0, 0',
	X = 1247.124  mm,	Y = -219.760  mm,	Z = -248.044  mm,
	W = 0.000 deg,	P = 30.000 deg,	R = -179.964 deg
};
P[258]{
   GP1:
	UF : 0, UT : 1,		CONFIG : 'N U T, 0, 0, 0',
	X = 1247.125  mm,	Y = -221.760  mm,	Z = -248.082  mm,
	W = 0.000 deg,	P = 30.000 deg,	R = -179.964 deg
};
P[259]{
   GP1:
	UF : 0, UT : 1,		CONFIG : 'N U T, 0, 0, 0',
	X = 1247.127  mm,	Y = -223.760  mm,	Z = -248.120  mm,
	W = 0.000 deg,	P = 30.000 deg,	R = -179.964 deg
};
P[260]{
   GP1:
	UF : 0, UT : 1,		CONFIG : 'N U T, 0, 0, 0',
	X = 1247.128  mm,	Y = -225.759  mm,	Z = -248.159  mm,
	W = 0.000 deg,	P = 30.000 deg,	R = -179.964 deg
};
P[261]{
   GP1:
	UF : 0, UT : 1,		CONFIG : 'N U T, 0, 0, 0',
	X = 1247.129  mm,	Y = -227.759  mm,	Z = -248.197  mm,
	W = 0.000 deg,	P = 30.000 deg,	R = -179.964 deg
};
P[262]{
   GP1:
	UF : 0, UT : 1,		CONFIG : 'N U T, 0, 0, 0',
	X = 1247.130  mm,	Y = -229.759  mm,	Z = -248.235  mm,
	W = 0.000 deg,	P = 30.000 deg,	R = -179.964 deg
};
P[263]{
   GP1:
	UF : 0, UT : 1,		CONFIG : 'N U T, 0, 0, 0',
	X = 1247.132  mm,	Y = -231.758  mm,	Z = -248.274  mm,
	W = 0.000 deg,	P = 30.000 deg,	R = -179.964 deg
};
P[264]{
   GP1:
	UF : 0, UT : 1,		CONFIG : 'N U T, 0, 0, 0',
	X = 1253.133  mm,	Y = -233.754  mm,	Z = -248.312  mm,
	W = 0.000 deg,	P = 30.000 deg,	R = -179.964 deg
};
P[265]{
   GP1:
	UF : 0, UT : 1,		CONFIG : 'N U T, 0, 0, 0',
	X = 1247.134  mm,	Y = -235.757  mm,	Z = -248.350  mm,
	W = 0.000 deg,	P = 30.000 deg,	R = -179.964 deg
};
P[266]{
   GP1:
	UF : 0, UT : 1,		CONFIG : 'N U T, 0, 0, 0',
	X = 1247.135  mm,	Y = -237.757  mm,	Z = -248.389  mm,
	W = 0.000 deg,	P = 30.000 deg,	R = -179.964 deg
};
P[267]{
   GP1:
	UF : 0, UT : 1,		CONFIG : 'N U T, 0, 0, 0',
	X = 1247.137  mm,	Y = -239.757  mm,	Z = -248.427  mm,
	W = 0.000 deg,	P = 30.000 deg,	R = -179.964 deg
};
P[268]{
   GP1:
	UF : 0, UT : 1,		CONFIG : 'N U T, 0, 0, 0',
	X = 1247.138  mm,	Y = -241.756  mm,	Z = -248.465  mm,
	W = 0.000 deg,	P = 30.000 deg,	R = 166.300 deg
};
P[269]{
   GP1:
	UF : 0, UT : 1,		CONFIG : 'N U T, 0, 0, 0',
	X = 1247.139  mm,	Y = -243.756  mm,	Z = -248.504  mm,
	W = 0.000 deg,	P = 30.000 deg,	R = 158.694 deg
};
P[270]{
   GP1:
	UF : 0, UT : 1,		CONFIG : 'N U T, 0, 0, 0',
	X = 1247.140  mm,	Y = -245.756  mm,	Z = -248.542  mm,
	W = 0.000 deg,	P = 30.000 deg,	R = 151.089 deg
};
P[271]{
   GP1:
	UF : 0, UT : 1,		CONFIG : 'N U T, 0, 0, 0',
	X = 1247.142  mm,	Y = -247.755  mm,	Z = -248.580  mm,
	W = 0.000 deg,	P = 30.000 deg,	R = 143.483 deg
};
P[272]{
   GP1:
	UF : 0, UT : 1,		CONFIG : 'N U T, 0, 0, 0',
	X = 1247.143  mm,	Y = -249.755  mm,	Z = -248.619  mm,
	W = 0.000 deg,	P = 30.000 deg,	R = 142.008 deg
};
P[273]{
   GP1:
	UF : 0, UT : 1,		CONFIG : 'N U T, 0, 0, 0',
	X = 1247.700  mm,	Y = -248.151  mm,	Z = -248.621  mm,
	W = 0.000 deg,	P = 30.000 deg,	R = 142.008 deg
};
P[274]{
   GP1:
	UF : 0, UT : 1,		CONFIG : 'N U T, 0, 0, 0',
	X = 1246.641  mm,	Y = -249.502  mm,	Z = -248.407  mm,
	W = 0.000 deg,	P = 30.000 deg,	R = 142.008 deg
};
P[275]{
   GP1:
	UF : 0, UT : 1,		CONFIG : 'N U T, 0, 0, 0',
	X = 1250.147  mm,	Y = -254.761  mm,	Z = -248.177  mm,
	W = 0.000 deg,	P = 30.000 deg,	R = 142.008 deg
};
P[276]{
   GP1:
	UF : 0, UT : 1,		CONFIG : 'N U T, 0, 0, 0',
	X = 1248.924  mm,	Y = -256.327  mm,	Z = -247.946  mm,
	W = 0.000 deg,	P = 30.000 deg,	R = 142.008 deg
};
P[277]{
   GP1:
	UF : 0, UT : 1,		CONFIG : 'N U T, 0, 0, 0',
	X = 1242.972  mm,	Y = -254.199  mm,	Z = -247.716  mm,
	W = 0.000 deg,	P = 30.000 deg,	R = 142.008 deg
};
P[278]{
   GP1:
	UF : 0, UT : 1,		CONFIG : 'N U T, 0, 0, 0',
	X = 1241.749  mm,	Y = -255.765  mm,	Z = -247.485  mm,
	W = 0.000 deg,	P = 30.000 deg,	R = 142.008 deg
};
P[279]{
   GP1:
	UF : 0, UT : 1,		CONFIG : 'N U T, 0, 0, 0',
	X = 1240.526  mm,	Y = -257.331  mm,	Z = -247.255  mm,
	W = 0.000 deg,	P = 30.000 deg,	R = 142.008 deg
};
P[280]{
   GP1:
	UF : 0, UT : 1,		CONFIG : 'N U T, 0, 0, 0',
	X = 1239.304  mm,	Y = -258.896  mm,	Z = -247.024  mm,
	W = 0.000 deg,	P = 30.000 deg,	R = 142.008 deg
};
P[281]{
   GP1:
	UF : 0, UT : 1,		CONFIG : 'N U T, 0, 0, 0',
	X = 1242.809  mm,	Y = -264.155  mm,	Z = -246.794  mm,
	W = 0.000 deg,	P = 30.000 deg,	R = 142.008 deg
};
P[282]{
   GP1:
	UF : 0, UT : 1,		CONFIG : 'N U T, 0, 0, 0',
	X = 1241.586  mm,	Y = -265.721  mm,	Z = -246.563  mm,
	W = 0.000 deg,	P = 30.000 deg,	R = 142.008 deg
};
P[283]{
   GP1:
	UF : 0, UT : 1,		CONFIG : 'N U T, 0, 0, 0',
	X = 1235.635  mm,	Y = -263.593  mm,	Z = -246.333  mm,
	W = 0.000 deg,	P = 30.000 deg,	R = 142.008 deg
};
P[284]{
   GP1:
	UF : 0, UT : 1,		CONFIG : 'N U T, 0, 0, 0',
	X = 1234.412  mm,	Y = -265.159  mm,	Z = -246.102  mm,
	W = 0.000 deg,	P = 30.000 deg,	R = 142.008 deg
};
P[285]{
   GP1:
	UF : 0, UT : 1,		CONFIG : 'N U T, 0, 0, 0',
	X = 1233.189  mm,	Y = -266.725  mm,	Z = -245.872  mm,
	W = 0.000 deg,	P = 30.000 deg,	R = 142.008 deg
};
P[286]{
   GP1:
	UF : 0, UT : 1,		CONFIG : 'N U T, 0, 0, 0',
	X = 1231.966  mm,	Y = -268.291  mm,	Z = -245.641  mm,
	W = 0.000 deg,	P = 30.000 deg,	R = 142.008 deg
};
P[287]{
   GP1:
	UF : 0, UT : 1,		CONFIG : 'N U T, 0, 0, 0',
	X = 1235.472  mm,	Y = -273.550  mm,	Z = -245.411  mm,
	W = 0.000 deg,	P = 30.000 deg,	R = 142.008 deg
};
P[288]{
   GP1:
	UF : 0, UT : 1,		CONFIG : 'N U T, 0, 0, 0',
	X = 1229.520  mm,	Y = -271.422  mm,	Z = -245.180  mm,
	W = 0.000 deg,	P = 30.000 deg,	R = 142.008 deg
};
P[289]{
   GP1:
	UF : 0, UT : 1,		CONFIG : 'N U T, 0, 0, 0',
	X = 1228.297  mm,	Y = -272.988  mm,	Z = -244.950  mm,
	W = 0.000 deg,	P = 30.000 deg,	R = 142.008 deg
};
P[290]{
   GP1:
	UF : 0, UT : 1,		CONFIG : 'N U T, 0, 0, 0',
	X = 1227.075  mm,	Y = -274.553  mm,	Z = -244.720  mm,
	W = 0.000 deg,	P = 30.000 deg,	R = 142.008 deg
};
P[291]{
   GP1:
	UF : 0, UT : 1,		CONFIG : 'N U T, 0, 0, 0',
	X = 1225.852  mm,	Y = -276.119  mm,	Z = -244.489  mm,
	W = 0.000 deg,	P = 30.000 deg,	R = 142.008 deg
};
P[292]{
   GP1:
	UF : 0, UT : 1,		CONFIG : 'N U T, 0, 0, 0',
	X = 1229.357  mm,	Y = -281.378  mm,	Z = -244.259  mm,
	W = 0.000 deg,	P = 30.000 deg,	R = 142.008 deg
};
P[293]{
   GP1:
	UF : 0, UT : 1,		CONFIG : 'N U T, 0, 0, 0',
	X = 1228.134  mm,	Y = -282.944  mm,	Z = -244.028  mm,
	W = 0.000 deg,	P = 30.000 deg,	R = 142.008 deg
};
P[294]{
   GP1:
	UF : 0, UT : 1,		CONFIG : 'N U T, 0, 0, 0',
	X = 1222.183  mm,	Y = -280.816  mm,	Z = -243.798  mm,
	W = 0.000 deg,	P = 30.000 deg,	R = 142.008 deg
};
P[295]{
   GP1:
	UF : 0, UT : 1,		CONFIG : 'N U T, 0, 0, 0',
	X = 1220.960  mm,	Y = -282.382  mm,	Z = -243.567  mm,
	W = 0.000 deg,	P = 30.000 deg,	R = 142.008 deg
};
P[296]{
   GP1:
	UF : 0, UT : 1,		CONFIG : 'N U T, 0, 0, 0',
	X = 1219.737  mm,	Y = -283.947  mm,	Z = -243.337  mm,
	W = 0.000 deg,	P = 30.000 deg,	R = 142.008 deg
};
P[297]{
   GP1:
	UF : 0, UT : 1,		CONFIG : 'N U T, 0, 0, 0',
	X = 1223.243  mm,	Y = -289.206  mm,	Z = -243.106  mm,
	W = 0.000 deg,	P = 30.000 deg,	R = 148.776 deg
};
P[298]{
   GP1:
	UF : 0, UT : 1,		CONFIG : 'N U T, 0, 0, 0',
	X = 1222.020  mm,	Y = -290.772  mm,	Z = -242.876  mm,
	W = 0.000 deg,	P = 30.000 deg,	R = 156.051 deg
};
P[299]{
   GP1:
	UF : 0, UT : 1,		CONFIG : 'N U T, 0, 0, 0',
	X = 1220.797  mm,	Y = -292.338  mm,	Z = -242.645  mm,
	W = 0.000 deg,	P = 30.000 deg,	R = 163.327 deg
};
P[300]{
   GP1:
	UF : 0, UT : 1,		CONFIG : 'N U T, 0, 0, 0',
	X = 1219.574  mm,	Y = -293.904  mm,	Z = -242.415  mm,
	W = 0.000 deg,	P = 30.000 deg,	R = 170.602 deg
};
P[301]{
   GP1:
	UF : 0, UT : 1,		CONFIG : 'N U T, 0, 0, 0',
	X = 1218.351  mm,	Y = -295.469  mm,	Z = -242.184  mm,
	W = 0.000 deg,	P = 30.000 deg,	R = 177.877 deg
};
P[302]{
   GP1:
	UF : 0, UT : 1,		CONFIG : 'N U T, 0, 0, 0',
	X = 1218.324  mm,	Y = -295.186  mm,	Z = -242.085  mm,
	W = 0.000 deg,	P = 30.000 deg,	R = 178.384 deg
};
P[303]{
   GP1:
	UF : 0, UT : 1,		CONFIG : 'N U T, 0, 0, 0',
	X = 1218.425  mm,	Y = -295.519  mm,	Z = -242.091  mm,
	W = 0.000 deg,	P = 30.000 deg,	R = 178.384 deg
};
P[304]{
   GP1:
	UF : 0, UT : 1,		CONFIG : 'N U T, 0, 0, 0',
	X = 1218.369  mm,	Y = -297.518  mm,	Z = -242.101  mm,
	W = 0.000 deg,	P = 30.000 deg,	R = 178.384 deg
};
P[305]{
   GP1:
	UF : 0, UT : 1,		CONFIG : 'N U T, 0, 0, 0',
	X = 1212.315  mm,	Y = -299.348  mm,	Z = -242.112  mm,
	W = 0.000 deg,	P = 30.000 deg,	R = 178.384 deg
};
P[306]{
   GP1:
	UF : 0, UT : 1,		CONFIG : 'N U T, 0, 0, 0',
	X = 1212.258  mm,	Y = -301.347  mm,	Z = -242.123  mm,
	W = 0.000 deg,	P = 30.000 deg,	R = 178.384 deg
};
P[307]{
   GP1:
	UF : 0, UT : 1,		CONFIG : 'N U T, 0, 0, 0',
	X = 1218.199  mm,	Y = -303.516  mm,	Z = -242.134  mm,
	W = 0.000 deg,	P = 30.000 deg,	R = 178.384 deg
};
P[308]{
   GP1:
	UF : 0, UT : 1,		CONFIG : 'N U T, 0, 0, 0',
	X = 1212.145  mm,	Y = -305.346  mm,	Z = -242.144  mm,
	W = 0.000 deg,	P = 30.000 deg,	R = 178.384 deg
};
P[309]{
   GP1:
	UF : 0, UT : 1,		CONFIG : 'N U T, 0, 0, 0',
	X = 1212.089  mm,	Y = -307.345  mm,	Z = -242.155  mm,
	W = 0.000 deg,	P = 30.000 deg,	R = 178.384 deg
};
P[310]{
   GP1:
	UF : 0, UT : 1,		CONFIG : 'N U T, 0, 0, 0',
	X = 1218.030  mm,	Y = -309.513  mm,	Z = -242.166  mm,
	W = 0.000 deg,	P = 30.000 deg,	R = 178.384 deg
};
P[311]{
   GP1:
	UF : 0, UT : 1,		CONFIG : 'N U T, 0, 0, 0',
	X = 1211.976  mm,	Y = -311.343  mm,	Z = -242.176  mm,
	W = 0.000 deg,	P = 30.000 deg,	R = 178.384 deg
};
P[312]{
   GP1:
	UF : 0, UT : 1,		CONFIG : 'N U T, 0, 0, 0',
	X = 1211.920  mm,	Y = -313.342  mm,	Z = -242.187  mm,
	W = 0.000 deg,	P = 30.000 deg,	R = 178.384 deg
};
P[313]{
   GP1:
	UF : 0, UT : 1,		CONFIG : 'N U T, 0, 0, 0',
	X = 1211.863  mm,	Y = -315.342  mm,	Z = -242.198  mm,
	W = 0.000 deg,	P = 30.000 deg,	R = 178.384 deg
};
P[314]{
   GP1:
	UF : 0, UT : 1,		CONFIG : 'N U T, 0, 0, 0',
	X = 1211.807  mm,	Y = -317.341  mm,	Z = -242.208  mm,
	W = 0.000 deg,	P = 30.000 deg,	R = 178.384 deg
};
P[315]{
   GP1:
	UF : 0, UT : 1,		CONFIG : 'N U T, 0, 0, 0',
	X = 1217.748  mm,	Y = -319.509  mm,	Z = -242.219  mm,
	W = 0.000 deg,	P = 30.000 deg,	R = 178.384 deg
};
P[316]{
   GP1:
	UF : 0, UT : 1,		CONFIG : 'N U T, 0, 0, 0',
	X = 1211.694  mm,	Y = -321.339  mm,	Z = -242.230  mm,
	W = 0.000 deg,	P = 30.000 deg,	R = 178.384 deg
};
P[317]{
   GP1:
	UF : 0, UT : 1,		CONFIG : 'N U T, 0, 0, 0',
	X = 1211.638  mm,	Y = -323.338  mm,	Z = -242.241  mm,
	W = 0.000 deg,	P = 30.000 deg,	R = 178.384 deg
};
P[318]{
   GP1:
	UF : 0, UT : 1,		CONFIG : 'N U T, 0, 0, 0',
	X = 1217.579  mm,	Y = -325.507  mm,	Z = -242.251  mm,
	W = 0.000 deg,	P = 30.000 deg,	R = 178.384 deg
};
P[319]{
   GP1:
	UF : 0, UT : 1,		CONFIG : 'N U T, 0, 0, 0',
	X = 1211.525  mm,	Y = -327.337  mm,	Z = -242.262  mm,
	W = 0.000 deg,	P = 30.000 deg,	R = 178.384 deg
};
P[320]{
   GP1:
	UF : 0, UT : 1,		CONFIG : 'N U T, 0, 0, 0',
	X = 1211.469  mm,	Y = -329.336  mm,	Z = -242.273  mm,
	W = 0.000 deg,	P = 30.000 deg,	R = 178.384 deg
};
P[321]{
   GP1:
	UF : 0, UT : 1,		CONFIG : 'N U T, 0, 0, 0',
	X = 1217.410  mm,	Y = -331.504  mm,	Z = -242.283  mm,
	W = 0.000 deg,	P = 30.000 deg,	R = 178.384 deg
};
P[322]{
   GP1:
	UF : 0, UT : 1,		CONFIG : 'N U T, 0, 0, 0',
	X = 1211.356  mm,	Y = -333.334  mm,	Z = -242.294  mm,
	W = 0.000 deg,	P = 30.000 deg,	R = 178.384 deg
};
P[323]{
   GP1:
	UF : 0, UT : 1,		CONFIG : 'N U T, 0, 0, 0',
	X = 1211.300  mm,	Y = -335.333  mm,	Z = -242.305  mm,
	W = 0.000 deg,	P = 30.000 deg,	R = 178.384 deg
};
P[324]{
   GP1:
	UF : 0, UT : 1,		CONFIG : 'N U T, 0, 0, 0',
	X = 1217.241  mm,	Y = -337.502  mm,	Z = -242.315  mm,
	W = 0.000 deg,	P = 30.000 deg,	R = 178.384 deg
};
P[325]{
   GP1:
	UF : 0, UT : 1,		CONFIG : 'N U T, 0, 0, 0',
	X = 1211.187  mm,	Y = -339.332  mm,	Z = -242.326  mm,
	W = 0.000 deg,	P = 30.000 deg,	R = 178.384 deg
};
P[326]{
   GP1:
	UF : 0, UT : 1,		CONFIG : 'N U T, 0, 0, 0',
	X = 1211.130  mm,	Y = -341.331  mm,	Z = -242.337  mm,
	W = 0.000 deg,	P = 30.000 deg,	R = 178.384 deg
};
P[327]{
   GP1:
	UF : 0, UT : 1,		CONFIG : 'N U T, 0, 0, 0',
	X = 1217.072  mm,	Y = -343.499  mm,	Z = -242.348  mm,
	W = 0.000 deg,	P = 30.000 deg,	R = 178.384 deg
};
P[328]{
   GP1:
	UF : 0, UT : 1,		CONFIG : 'N U T, 0, 0, 0',
	X = 1211.018  mm,	Y = -345.329  mm,	Z = -242.358  mm,
	W = 0.000 deg,	P = 30.000 deg,	R = 178.384 deg
};
P[329]{
   GP1:
	UF : 0, UT : 1,		CONFIG : 'N U T, 0, 0, 0',
	X = 1210.961  mm,	Y = -347.328  mm,	Z = -242.369  mm,
	W = 0.000 deg,	P = 30.000 deg,	R = 178.384 deg
};
P[330]{
   GP1:
	UF : 0, UT : 1,		CONFIG : 'N U T, 0, 0, 0',
	X = 1210.905  mm,	Y = -349.328  mm,	Z = -242.380  mm,
	W = 0.000 deg,	P = 30.000 deg,	R = 178.384 deg
};
P[331]{
   GP1:
	UF : 0, UT : 1,		CONFIG : 'N U T, 0, 0, 0',
	X = 1210.848  mm,	Y = -351.327  mm,	Z = -242.390  mm,
	W = 0.000 deg,	P = 30.000 deg,	R = 178.384 deg
};
P[332]{
   GP1:
	UF : 0, UT : 1,		CONFIG : 'N U T, 0, 0, 0',
	X = 1216.790  mm,	Y = -353.495  mm,	Z = -242.401  mm,
	W = 0.000 deg,	P = 30.000 deg,	R = 178.384 deg
};
P[333]{
   GP1:
	UF : 0, UT : 1,		CONFIG : 'N U T, 0, 0, 0',
	X = 1210.736  mm,	Y = -355.325  mm,	Z = -242.412  mm,
	W = 0.000 deg,	P = 30.000 deg,	R = 178.384 deg
};
P[334]{
   GP1:
	UF : 0, UT : 1,		CONFIG : 'N U T, 0, 0, 0',
	X = 1210.679  mm,	Y = -357.324  mm,	Z = -242.422  mm,
	W = 0.000 deg,	P = 30.000 deg,	R = 178.384 deg
};
P[335]{
   GP1:
	UF : 0, UT : 1,		CONFIG : 'N U T, 0, 0, 0',
	X = 1216.620  mm,	Y = -359.493  mm,	Z = -242.433  mm,
	W = 0.000 deg,	P = 30.000 deg,	R = -169.630 deg
};
P[336]{
   GP1:
	UF : 0, UT : 1,		CONFIG : 'N U T, 0, 0, 0',
	X = 1216.564  mm,	Y = -361.492  mm,	Z = -242.444  mm,
	W = 0.000 deg,	P = 30.000 deg,	R = -161.985 deg
};
P[337]{
   GP1:
	UF : 0, UT : 1,		CONFIG : 'N U T, 0, 0, 0',
	X = 1216.508  mm,	Y = -363.491  mm,	Z = -242.455  mm,
	W = 0.000 deg,	P = 30.000 deg,	R = -154.340 deg
};
P[338]{
   GP1:
	UF : 0, UT : 1,		CONFIG : 'N U T, 0, 0, 0',
	X = 1216.451  mm,	Y = -365.490  mm,	Z = -242.465  mm,
	W = 0.000 deg,	P = 30.000 deg,	R = -146.695 deg
};
P[339]{
   GP1:
	UF : 0, UT : 1,		CONFIG : 'N U T, 0, 0, 0',
	X = 1216.314  mm,	Y = -365.710  mm,	Z = -242.471  mm,
	W = 0.000 deg,	P = 30.000 deg,	R = -143.390 deg
};
P[340]{
   GP1:
	UF : 0, UT : 1,		CONFIG : 'N U T, 0, 0, 0',
	X = 1216.361  mm,	Y = -365.433  mm,	Z = -242.588  mm,
	W = 0.000 deg,	P = 30.000 deg,	R = -143.390 deg
};
P[341]{
   GP1:
	UF : 0, UT : 1,		CONFIG : 'N U T, 0, 0, 0',
	X = 1212.727  mm,	Y = -370.602  mm,	Z = -242.850  mm,
	W = 0.000 deg,	P = 30.000 deg,	R = -143.390 deg
};
P[342]{
   GP1:
	UF : 0, UT : 1,		CONFIG : 'N U T, 0, 0, 0',
	X = 1213.909  mm,	Y = -372.194  mm,	Z = -243.111  mm,
	W = 0.000 deg,	P = 30.000 deg,	R = -143.390 deg
};
P[343]{
   GP1:
	UF : 0, UT : 1,		CONFIG : 'N U T, 0, 0, 0',
	X = 1215.092  mm,	Y = -373.786  mm,	Z = -243.372  mm,
	W = 0.000 deg,	P = 30.000 deg,	R = -143.390 deg
};
P[344]{
   GP1:
	UF : 0, UT : 1,		CONFIG : 'N U T, 0, 0, 0',
	X = 1216.274  mm,	Y = -375.377  mm,	Z = -243.633  mm,
	W = 0.000 deg,	P = 30.000 deg,	R = -143.390 deg
};
P[345]{
   GP1:
	UF : 0, UT : 1,		CONFIG : 'N U T, 0, 0, 0',
	X = 1222.273  mm,	Y = -373.391  mm,	Z = -243.894  mm,
	W = 0.000 deg,	P = 30.000 deg,	R = -143.390 deg
};
P[346]{
   GP1:
	UF : 0, UT : 1,		CONFIG : 'N U T, 0, 0, 0',
	X = 1223.456  mm,	Y = -374.983  mm,	Z = -244.155  mm,
	W = 0.000 deg,	P = 30.000 deg,	R = -143.390 deg
};
P[347]{
   GP1:
	UF : 0, UT : 1,		CONFIG : 'N U T, 0, 0, 0',
	X = 1224.638  mm,	Y = -376.574  mm,	Z = -244.417  mm,
	W = 0.000 deg,	P = 30.000 deg,	R = -143.390 deg
};
P[348]{
   GP1:
	UF : 0, UT : 1,		CONFIG : 'N U T, 0, 0, 0',
	X = 1221.004  mm,	Y = -381.744  mm,	Z = -244.678  mm,
	W = 0.000 deg,	P = 30.000 deg,	R = -143.390 deg
};
P[349]{
   GP1:
	UF : 0, UT : 1,		CONFIG : 'N U T, 0, 0, 0',
	X = 1222.187  mm,	Y = -383.336  mm,	Z = -244.939  mm,
	W = 0.000 deg,	P = 30.000 deg,	R = -143.390 deg
};
P[350]{
   GP1:
	UF : 0, UT : 1,		CONFIG : 'N U T, 0, 0, 0',
	X = 1223.369  mm,	Y = -384.928  mm,	Z = -245.200  mm,
	W = 0.000 deg,	P = 30.000 deg,	R = -143.390 deg
};
P[351]{
   GP1:
	UF : 0, UT : 1,		CONFIG : 'N U T, 0, 0, 0',
	X = 1224.552  mm,	Y = -386.519  mm,	Z = -245.461  mm,
	W = 0.000 deg,	P = 30.000 deg,	R = -143.390 deg
};
P[352]{
   GP1:
	UF : 0, UT : 1,		CONFIG : 'N U T, 0, 0, 0',
	X = 1225.734  mm,	Y = -388.111  mm,	Z = -245.723  mm,
	W = 0.000 deg,	P = 30.000 deg,	R = -143.390 deg
};
P[353]{
   GP1:
	UF : 0, UT : 1,		CONFIG : 'N U T, 0, 0, 0',
	X = 1226.917  mm,	Y = -389.703  mm,	Z = -245.984  mm,
	W = 0.000 deg,	P = 30.000 deg,	R = -143.390 deg
};
P[354]{
   GP1:
	UF : 0, UT : 1,		CONFIG : 'N U T, 0, 0, 0',
	X = 1232.916  mm,	Y = -387.716  mm,	Z = -246.245  mm,
	W = 0.000 deg,	P = 30.000 deg,	R = -143.390 deg
};
P[355]{
   GP1:
	UF : 0, UT : 1,		CONFIG : 'N U T, 0, 0, 0',
	X = 1234.098  mm,	Y = -389.308  mm,	Z = -246.506  mm,
	W = 0.000 deg,	P = 30.000 deg,	R = -143.390 deg
};
P[356]{
   GP1:
	UF : 0, UT : 1,		CONFIG : 'N U T, 0, 0, 0',
	X = 1230.465  mm,	Y = -394.478  mm,	Z = -246.767  mm,
	W = 0.000 deg,	P = 30.000 deg,	R = -143.390 deg
};
P[357]{
   GP1:
	UF : 0, UT : 1,		CONFIG : 'N U T, 0, 0, 0',
	X = 1231.647  mm,	Y = -396.069  mm,	Z = -247.028  mm,
	W = 0.000 deg,	P = 30.000 deg,	R = -143.390 deg
};
P[358]{
   GP1:
	UF : 0, UT : 1,		CONFIG : 'N U T, 0, 0, 0',
	X = 1232.830  mm,	Y = -397.661  mm,	Z = -247.290  mm,
	W = 0.000 deg,	P = 30.000 deg,	R = -143.390 deg
};
P[359]{
   GP1:
	UF : 0, UT : 1,		CONFIG : 'N U T, 0, 0, 0',
	X = 1234.012  mm,	Y = -399.253  mm,	Z = -247.551  mm,
	W = 0.000 deg,	P = 30.000 deg,	R = -143.390 deg
};
P[360]{
   GP1:
	UF : 0, UT : 1,		CONFIG : 'N U T, 0, 0, 0',
	X = 1240.011  mm,	Y = -397.266  mm,	Z = -247.812  mm,
	W = 0.000 deg,	P = 30.000 deg,	R = -143.390 deg
};
P[361]{
   GP1:
	UF : 0, UT : 1,		CONFIG : 'N U T, 0, 0, 0',
	X = 1241.193  mm,	Y = -398.858  mm,	Z = -248.073  mm,
	W = 0.000 deg,	P = 30.000 deg,	R = -143.390 deg
};
P[362]{
   GP1:
	UF : 0, UT : 1,		CONFIG : 'N U T, 0, 0, 0',
	X = 1237.560  mm,	Y = -404.028  mm,	Z = -248.334  mm,
	W = 0.000 deg,	P = 30.000 deg,	R = -146.704 deg
};
P[363]{
   GP1:
	UF : 0, UT : 1,		CONFIG : 'N U T, 0, 0, 0',
	X = 1238.742  mm,	Y = -405.619  mm,	Z = -248.595  mm,
	W = 0.000 deg,	P = 30.000 deg,	R = -154.082 deg
};
P[364]{
   GP1:
	UF : 0, UT : 1,		CONFIG : 'N U T, 0, 0, 0',
	X = 1239.925  mm,	Y = -407.211  mm,	Z = -248.857  mm,
	W = 0.000 deg,	P = 30.000 deg,	R = -161.460 deg
};
P[365]{
   GP1:
	UF : 0, UT : 1,		CONFIG : 'N U T, 0, 0, 0',
	X = 1241.107  mm,	Y = -408.803  mm,	Z = -249.118  mm,
	W = 0.000 deg,	P = 30.000 deg,	R = -168.839 deg
};
P[366]{
   GP1:
	UF : 0, UT : 1,		CONFIG : 'N U T, 0, 0, 0',
	X = 1242.290  mm,	Y = -410.394  mm,	Z = -249.379  mm,
	W = 0.000 deg,	P = 30.000 deg,	R = -176.217 deg
};
P[367]{
   GP1:
	UF : 0, UT : 1,		CONFIG : 'N U T, 0, 0, 0',
	X = 1243.472  mm,	Y = -411.986  mm,	Z = -249.640  mm,
	W = 0.000 deg,	P = 30.000 deg,	R = 179.719 deg
};
P[368]{
   GP1:
	UF : 0, UT : 1,		CONFIG : 'N U T, 0, 0, 0',
	X = 1242.946  mm,	Y = -410.368  mm,	Z = -249.654  mm,
	W = 0.000 deg,	P = 30.000 deg,	R = 179.719 deg
};
P[369]{
   GP1:
	UF : 0, UT : 1,		CONFIG : 'N U T, 0, 0, 0',
	X = 1242.936  mm,	Y = -412.160  mm,	Z = -249.677  mm,
	W = 0.000 deg,	P = 30.000 deg,	R = 179.719 deg
};
P[370]{
   GP1:
	UF : 0, UT : 1,		CONFIG : 'N U T, 0, 0, 0',
	X = 1248.926  mm,	Y = -414.189  mm,	Z = -249.701  mm,
	W = 0.000 deg,	P = 30.000 deg,	R = 179.719 deg
};
P[371]{
   GP1:
	UF : 0, UT : 1,		CONFIG : 'N U T, 0, 0, 0',
	X = 1248.916  mm,	Y = -416.189  mm,	Z = -249.724  mm,
	W = 0.000 deg,	P = 30.000 deg,	R = 179.719 deg
};
P[372]{
   GP1:
	UF : 0, UT : 1,		CONFIG : 'N U T, 0, 0, 0',
	X = 1248.906  mm,	Y = -418.189  mm,	Z = -249.748  mm,
	W = 0.000 deg,	P = 30.000 deg,	R = 179.719 deg
};
P[373]{
   GP1:
	UF : 0, UT : 1,		CONFIG : 'N U T, 0, 0, 0',
	X = 1248.896  mm,	Y = -420.189  mm,	Z = -249.772  mm,
	W = 0.000 deg,	P = 30.000 deg,	R = 179.719 deg
};
P[374]{
   GP1:
	UF : 0, UT : 1,		CONFIG : 'N U T, 0, 0, 0',
	X = 1242.887  mm,	Y = -422.159  mm,	Z = -249.796  mm,
	W = 0.000 deg,	P = 30.000 deg,	R = 179.719 deg
};
P[375]{
   GP1:
	UF : 0, UT : 1,		CONFIG : 'N U T, 0, 0, 0',
	X = 1248.877  mm,	Y = -424.188  mm,	Z = -249.819  mm,
	W = 0.000 deg,	P = 30.000 deg,	R = 179.719 deg
};
P[376]{
   GP1:
	UF : 0, UT : 1,		CONFIG : 'N U T, 0, 0, 0',
	X = 1248.867  mm,	Y = -426.188  mm,	Z = -249.843  mm,
	W = 0.000 deg,	P = 30.000 deg,	R = 179.719 deg
};
P[377]{
   GP1:
	UF : 0, UT : 1,		CONFIG : 'N U T, 0, 0, 0',
	X = 1242.857  mm,	Y = -428.159  mm,	Z = -249.867  mm,
	W = 0.000 deg,	P = 30.000 deg,	R = 179.719 deg
};
P[378]{
   GP1:
	UF : 0, UT : 1,		CONFIG : 'N U T, 0, 0, 0',
	X = 1248.847  mm,	Y = -430.188  mm,	Z = -249.891  mm,
	W = 0.000 deg,	P = 30.000 deg,	R = 179.719 deg
};
P[379]{
   GP1:
	UF : 0, UT : 1,		CONFIG : 'N U T, 0, 0, 0',
	X = 1248.838  mm,	Y = -432.188  mm,	Z = -249.914  mm,
	W = 0.000 deg,	P = 30.000 deg,	R = 179.719 deg
};
P[380]{
   GP1:
	UF : 0, UT : 1,		CONFIG : 'N U T, 0, 0, 0',
	X = 1248.828  mm,	Y = -434.187  mm,	Z = -249.938  mm,
	W = 0.000 deg,	P = 30.000 deg,	R = 179.719 deg
};
P[381]{
   GP1:
	UF : 0, UT : 1,		CONFIG : 'N U T, 0, 0, 0',
	X = 1248.818  mm,	Y = -436.187  mm,	Z = -249.962  mm,
	W = 0.000 deg,	P = 30.000 deg,	R = 179.719 deg
};
P[382]{
   GP1:
	UF : 0, UT : 1,		CONFIG : 'N U T, 0, 0, 0',
	X = 1242.808  mm,	Y = -438.158  mm,	Z = -249.986  mm,
	W = 0.000 deg,	P = 30.000 deg,	R = 179.719 deg
};
P[383]{
   GP1:
	UF : 0, UT : 1,		CONFIG : 'N U T, 0, 0, 0',
	X = 1248.798  mm,	Y = -440.187  mm,	Z = -250.009  mm,
	W = 0.000 deg,	P = 30.000 deg,	R = 179.719 deg
};
P[384]{
   GP1:
	UF : 0, UT : 1,		CONFIG : 'N U T, 0, 0, 0',
	X = 1248.789  mm,	Y = -442.187  mm,	Z = -250.033  mm,
	W = 0.000 deg,	P = 30.000 deg,	R = 179.719 deg
};
P[385]{
   GP1:
	UF : 0, UT : 1,		CONFIG : 'N U T, 0, 0, 0',
	X = 1248.779  mm,	Y = -444.187  mm,	Z = -250.057  mm,
	W = 0.000 deg,	P = 30.000 deg,	R = 179.719 deg
};
P[386]{
   GP1:
	UF : 0, UT : 1,		CONFIG : 'N U T, 0, 0, 0',
	X = 1248.769  mm,	Y = -446.186  mm,	Z = -250.081  mm,
	W = 0.000 deg,	P = 30.000 deg,	R = 179.719 deg
};
P[387]{
   GP1:
	UF : 0, UT : 1,		CONFIG : 'N U T, 0, 0, 0',
	X = 1242.759  mm,	Y = -448.157  mm,	Z = -250.104  mm,
	W = 0.000 deg,	P = 30.000 deg,	R = 179.719 deg
};
P[388]{
   GP1:
	UF : 0, UT : 1,		CONFIG : 'N U T, 0, 0, 0',
	X = 1248.749  mm,	Y = -450.186  mm,	Z = -250.128  mm,
	W = 0.000 deg,	P = 30.000 deg,	R = 179.719 deg
};
P[389]{
   GP1:
	UF : 0, UT : 1,		CONFIG : 'N U T, 0, 0, 0',
	X = 1248.740  mm,	Y = -452.186  mm,	Z = -250.152  mm,
	W = 0.000 deg,	P = 30.000 deg,	R = 179.719 deg
};
P[390]{
   GP1:
	UF : 0, UT : 1,		CONFIG : 'N U T, 0, 0, 0',
	X = 1242.730  mm,	Y = -454.156  mm,	Z = -250.176  mm,
	W = 0.000 deg,	P = 30.000 deg,	R = 179.719 deg
};
P[391]{
   GP1:
	UF : 0, UT : 1,		CONFIG : 'N U T, 0, 0, 0',
	X = 1248.720  mm,	Y = -456.186  mm,	Z = -250.200  mm,
	W = 0.000 deg,	P = 30.000 deg,	R = 179.719 deg
};
P[392]{
   GP1:
	UF : 0, UT : 1,		CONFIG : 'N U T, 0, 0, 0',
	X = 1248.710  mm,	Y = -458.185  mm,	Z = -250.223  mm,
	W = 0.000 deg,	P = 30.000 deg,	R = 179.719 deg
};
P[393]{
   GP1:
	UF : 0, UT : 1,		CONFIG : 'N U T, 0, 0, 0',
	X = 1248.700  mm,	Y = -460.185  mm,	Z = -250.247  mm,
	W = 0.000 deg,	P = 30.000 deg,	R = 179.719 deg
};
P[394]{
   GP1:
	UF : 0, UT : 1,		CONFIG : 'N U T, 0, 0, 0',
	X = 1248.691  mm,	Y = -462.185  mm,	Z = -250.271  mm,
	W = 0.000 deg,	P = 30.000 deg,	R = 179.719 deg
};
P[395]{
   GP1:
	UF : 0, UT : 1,		CONFIG : 'N U T, 0, 0, 0',
	X = 1242.681  mm,	Y = -464.156  mm,	Z = -250.295  mm,
	W = 0.000 deg,	P = 30.000 deg,	R = 179.719 deg
};
P[396]{
   GP1:
	UF : 0, UT : 1,		CONFIG : 'N U T, 0, 0, 0',
	X = 1248.671  mm,	Y = -466.185  mm,	Z = -250.318  mm,
	W = 0.000 deg,	P = 30.000 deg,	R = 179.719 deg
};
P[397]{
   GP1:
	UF : 0, UT : 1,		CONFIG : 'N U T, 0, 0, 0',
	X = 1248.661  mm,	Y = -468.185  mm,	Z = -250.342  mm,
	W = 0.000 deg,	P = 30.000 deg,	R = 179.719 deg
};
P[398]{
   GP1:
	UF : 0, UT : 1,		CONFIG : 'N U T, 0, 0, 0',
	X = 1242.651  mm,	Y = -470.155  mm,	Z = -250.366  mm,
	W = 0.000 deg,	P = 30.000 deg,	R = 172.305 deg
};
P[399]{
   GP1:
	UF : 0, UT : 1,		CONFIG : 'N U T, 0, 0, 0',
	X = 1242.642  mm,	Y = -472.155  mm,	Z = -250.390  mm,
	W = 0.000 deg,	P = 30.000 deg,	R = 164.463 deg
};
P[400]{
   GP1:
	UF : 0, UT : 1,		CONFIG : 'N U T, 0, 0, 0',
	X = 1242.632  mm,	Y = -474.155  mm,	Z = -250.413  mm,
	W = 0.000 deg,	P = 30.000 deg,	R = 156.621 deg
};
P[401]{
   GP1:
	UF : 0, UT : 1,		CONFIG : 'N U T, 0, 0, 0',
	X = 1242.622  mm,	Y = -476.155  mm,	Z = -250.437  mm,
	W = 0.000 deg,	P = 30.000 deg,	R = 148.779 deg
};
P[402]{
   GP1:
	UF : 0, UT : 1,		CONFIG : 'N U T, 0, 0, 0',
	X = 1242.612  mm,	Y = -478.154  mm,	Z = -250.461  mm,
	W = 0.000 deg,	P = 30.000 deg,	R = 140.937 deg
};
P[403]{
   GP1:
	UF : 0, UT : 1,		CONFIG : 'N U T, 0, 0, 0',
	X = 1242.995  mm,	Y = -477.228  mm,	Z = -250.467  mm,
	W = 0.000 deg,	P = 30.000 deg,	R = 140.509 deg
};
P[404]{
   GP1:
	UF : 0, UT : 1,		CONFIG : 'N U T, 0, 0, 0',
	X = 1246.996  mm,	Y = -481.733  mm,	Z = -250.288  mm,
	W = 0.000 deg,	P = 30.000 deg,	R = 140.509 deg
};
P[405]{
   GP1:
	UF : 0, UT : 1,		CONFIG : 'N U T, 0, 0, 0',
	X = 1245.734  mm,	Y = -483.265  mm,	Z = -250.044  mm,
	W = 0.000 deg,	P = 30.000 deg,	R = 140.509 deg
};
P[406]{
   GP1:
	UF : 0, UT : 1,		CONFIG : 'N U T, 0, 0, 0',
	X = 1244.471  mm,	Y = -484.797  mm,	Z = -249.801  mm,
	W = 0.000 deg,	P = 30.000 deg,	R = 140.509 deg
};
P[407]{
   GP1:
	UF : 0, UT : 1,		CONFIG : 'N U T, 0, 0, 0',
	X = 1243.209  mm,	Y = -486.329  mm,	Z = -249.557  mm,
	W = 0.000 deg,	P = 30.000 deg,	R = 140.509 deg
};
P[408]{
   GP1:
	UF : 0, UT : 1,		CONFIG : 'N U T, 0, 0, 0',
	X = 1237.316  mm,	Y = -484.045  mm,	Z = -249.314  mm,
	W = 0.000 deg,	P = 30.000 deg,	R = 140.509 deg
};
P[409]{
   GP1:
	UF : 0, UT : 1,		CONFIG : 'N U T, 0, 0, 0',
	X = 1240.684  mm,	Y = -489.392  mm,	Z = -249.070  mm,
	W = 0.000 deg,	P = 30.000 deg,	R = 140.509 deg
};
P[410]{
   GP1:
	UF : 0, UT : 1,		CONFIG : 'N U T, 0, 0, 0',
	X = 1239.421  mm,	Y = -490.924  mm,	Z = -248.827  mm,
	W = 0.000 deg,	P = 30.000 deg,	R = 140.509 deg
};
P[411]{
   GP1:
	UF : 0, UT : 1,		CONFIG : 'N U T, 0, 0, 0',
	X = 1233.529  mm,	Y = -488.641  mm,	Z = -248.583  mm,
	W = 0.000 deg,	P = 30.000 deg,	R = 140.509 deg
};
P[412]{
   GP1:
	UF : 0, UT : 1,		CONFIG : 'N U T, 0, 0, 0',
	X = 1232.266  mm,	Y = -490.173  mm,	Z = -248.340  mm,
	W = 0.000 deg,	P = 30.000 deg,	R = 140.509 deg
};
P[413]{
   GP1:
	UF : 0, UT : 1,		CONFIG : 'N U T, 0, 0, 0',
	X = 1235.634  mm,	Y = -495.520  mm,	Z = -248.096  mm,
	W = 0.000 deg,	P = 30.000 deg,	R = 140.509 deg
};
P[414]{
   GP1:
	UF : 0, UT : 1,		CONFIG : 'N U T, 0, 0, 0',
	X = 1234.372  mm,	Y = -497.052  mm,	Z = -247.853  mm,
	W = 0.000 deg,	P = 30.000 deg,	R = 140.509 deg
};
P[415]{
   GP1:
	UF : 0, UT : 1,		CONFIG : 'N U T, 0, 0, 0',
	X = 1228.479  mm,	Y = -494.768  mm,	Z = -247.609  mm,
	W = 0.000 deg,	P = 30.000 deg,	R = 140.509 deg
};
P[416]{
   GP1:
	UF : 0, UT : 1,		CONFIG : 'N U T, 0, 0, 0',
	X = 1231.847  mm,	Y = -500.116  mm,	Z = -247.366  mm,
	W = 0.000 deg,	P = 30.000 deg,	R = 140.509 deg
};
P[417]{
   GP1:
	UF : 0, UT : 1,		CONFIG : 'N U T, 0, 0, 0',
	X = 1230.584  mm,	Y = -501.648  mm,	Z = -247.122  mm,
	W = 0.000 deg,	P = 30.000 deg,	R = 140.509 deg
};
P[418]{
   GP1:
	UF : 0, UT : 1,		CONFIG : 'N U T, 0, 0, 0',
	X = 1229.322  mm,	Y = -503.180  mm,	Z = -246.878  mm,
	W = 0.000 deg,	P = 30.000 deg,	R = 140.509 deg
};
P[419]{
   GP1:
	UF : 0, UT : 1,		CONFIG : 'N U T, 0, 0, 0',
	X = 1228.059  mm,	Y = -504.712  mm,	Z = -246.635  mm,
	W = 0.000 deg,	P = 30.000 deg,	R = 140.509 deg
};
P[420]{
   GP1:
	UF : 0, UT : 1,		CONFIG : 'N U T, 0, 0, 0',
	X = 1222.167  mm,	Y = -502.428  mm,	Z = -246.391  mm,
	W = 0.000 deg,	P = 30.000 deg,	R = 140.509 deg
};
P[421]{
   GP1:
	UF : 0, UT : 1,		CONFIG : 'N U T, 0, 0, 0',
	X = 1225.534  mm,	Y = -507.776  mm,	Z = -246.148  mm,
	W = 0.000 deg,	P = 30.000 deg,	R = 140.509 deg
};
P[422]{
   GP1:
	UF : 0, UT : 1,		CONFIG : 'N U T, 0, 0, 0',
	X = 1224.272  mm,	Y = -509.308  mm,	Z = -245.904  mm,
	W = 0.000 deg,	P = 30.000 deg,	R = 140.509 deg
};
P[423]{
   GP1:
	UF : 0, UT : 1,		CONFIG : 'N U T, 0, 0, 0',
	X = 1218.379  mm,	Y = -507.024  mm,	Z = -245.661  mm,
	W = 0.000 deg,	P = 30.000 deg,	R = 140.509 deg
};
P[424]{
   GP1:
	UF : 0, UT : 1,		CONFIG : 'N U T, 0, 0, 0',
	X = 1217.117  mm,	Y = -508.556  mm,	Z = -245.417  mm,
	W = 0.000 deg,	P = 30.000 deg,	R = 140.509 deg
};
P[425]{
   GP1:
	UF : 0, UT : 1,		CONFIG : 'N U T, 0, 0, 0',
	X = 1220.485  mm,	Y = -513.904  mm,	Z = -245.174  mm,
	W = 0.000 deg,	P = 30.000 deg,	R = 144.040 deg
};
P[426]{
   GP1:
	UF : 0, UT : 1,		CONFIG : 'N U T, 0, 0, 0',
	X = 1219.222  mm,	Y = -515.436  mm,	Z = -244.930  mm,
	W = 0.000 deg,	P = 30.000 deg,	R = 148.841 deg
};
P[427]{
   GP1:
	UF : 0, UT : 1,		CONFIG : 'N U T, 0, 0, 0',
	X = 1217.960  mm,	Y = -516.968  mm,	Z = -244.687  mm,
	W = 0.000 deg,	P = 30.000 deg,	R = 153.642 deg
};
P[428]{
   GP1:
	UF : 0, UT : 1,		CONFIG : 'N U T, 0, 0, 0',
	X = 1216.697  mm,	Y = -518.500  mm,	Z = -244.443  mm,
	W = 0.000 deg,	P = 30.000 deg,	R = 158.443 deg
};
P[429]{
   GP1:
	UF : 0, UT : 1,		CONFIG : 'N U T, 0, 0, 0',
	X = 1215.435  mm,	Y = -520.032  mm,	Z = -244.200  mm,
	W = 0.000 deg,	P = 30.000 deg,	R = 163.244 deg
};
P[430]{
   GP1:
	UF : 0, UT : 1,		CONFIG : 'N U T, 0, 0, 0',
	X = 1214.656  mm,	Y = -520.977  mm,	Z = -244.049  mm,
	W = 0.000 deg,	P = 30.000 deg,	R = 164.514 deg
};
/END
